// TIA Portal project "FactoryIO_Template_S7-1200_V15_V16" (V16)
// Vorlageprojekt für das Buch mit Zielsystem S7-1200

(* hardware
DEVICE "S7-1200-Station_1"  S7-1200 Station
   slot 0: "Baugruppenträger_0"  Rack  V1.0
   slot 1: "PLC_1"  CPU 1214C DC/DC/Rly  6ES7 214-1HG40-0XB0  V4.4
   slot 2: "DQ 16x24VDC_1"  SM 1222 DQ16 x 24VDC  6ES7 222-1BH32-0XB0  V2.0
   slot 3: "DQ 16x24VDC_2"  SM 1222 DQ16 x 24VDC  6ES7 222-1BH32-0XB0  V2.0
   slot 4: "DQ 16x24VDC_3"  SM 1222 DQ16 x 24VDC  6ES7 222-1BH32-0XB0  V2.0
   slot 5: "DQ 16x24VDC_4"  SM 1222 DQ16 x 24VDC  6ES7 222-1BH32-0XB0  V2.0
   slot 6: "DQ 16x24VDC_5"  SM 1222 DQ16 x 24VDC  6ES7 222-1BH32-0XB0  V2.0
   slot 7: "DQ 16x24VDC_6"  SM 1222 DQ16 x 24VDC  6ES7 222-1BH32-0XB0  V2.0
   slot 8: "DQ 16x24VDC_7"  SM 1222 DQ16 x 24VDC  6ES7 222-1BH32-0XB0  V2.0
   slot 9: "DQ 16x24VDC_8"  SM 1222 DQ16 x 24VDC  6ES7 222-1BH32-0XB0  V2.0
*)

// ===== PLC "PLC_1"  CPU 1214C DC/DC/Rly =====

VAR_GLOBAL   // PLC tag table "Standard-Variablentabelle"
   "System" AT %M0.0 : Bool;
   "Blue Lids at Place Memory" AT %M0.1 : Bool;
   "Blue Bases at Place Memory" AT %M0.2 : Bool;
   "Blue S1" AT %M0.3 : Bool;
   "Blue S2" AT %M0.4 : Bool;
   "Blue S3" AT %M0.5 : Bool;
   "Blue S4" AT %M0.6 : Bool;
   "Blue S5" AT %M0.7 : Bool;
   "Blue S6" AT %M1.0 : Bool;
   "Blue S7" AT %M1.1 : Bool;
   "Blue S8" AT %M1.2 : Bool;
   "Blue S9" AT %M1.3 : Bool;
   "Blue S10" AT %M1.4 : Bool;
   "Blue S11" AT %M1.5 : Bool;
   "Green Lid at place memory" AT %M2.0 : Bool;
   "Green bases at place memory" AT %M2.1 : Bool;
   "Green S1" AT %M2.2 : Bool;
   "Green S2" AT %M2.3 : Bool;
   "Green S3" AT %M2.4 : Bool;
   "Green S4" AT %M2.5 : Bool;
   "Green S5" AT %M2.6 : Bool;
   "Green S6" AT %M2.7 : Bool;
   "Green S7" AT %M3.0 : Bool;
   "Green S8" AT %M3.1 : Bool;
   "Green S9" AT %M3.2 : Bool;
   "Green S10" AT %M3.3 : Bool;
   "Green S11" AT %M3.4 : Bool;
   "Metal S1" AT %M3.5 : Bool;
   "Metal S2" AT %M3.6 : Bool;
   "Metal S3" AT %M3.7 : Bool;
   "Metal S4" AT %M4.0 : Bool;
   "Metal S5" AT %M4.1 : Bool;
   "Metal S6" AT %M4.2 : Bool;
   "Metal S7" AT %M4.3 : Bool;
   "Metal S8" AT %M4.4 : Bool;
   "Metal S9" AT %M4.5 : Bool;
   "Metal S10" AT %M4.6 : Bool;
   "Metal S11" AT %M4.7 : Bool;
   "Metal Lid at place memory" AT %M5.0 : Bool;
   "Metal bases at place memory" AT %M5.1 : Bool;
   "Blue Pallet lid at place memory" AT %M5.2 : Bool;
   "Blue Pallet bases at place memory" AT %M5.3 : Bool;
   "Blue Pallet S1" AT %M5.4 : Bool;
   "Blue Pallet S2" AT %M5.5 : Bool;
   "Blue Pallet S3" AT %M5.6 : Bool;
   "Blue Pallet S4" AT %M5.7 : Bool;
   "Blue Pallet S5" AT %M6.0 : Bool;
   "Blue Pallet S6" AT %M6.1 : Bool;
   "Blue Pallet S7" AT %M6.2 : Bool;
   "Blue Pallet S8" AT %M6.3 : Bool;
   "Blue Pallet S9" AT %M6.4 : Bool;
   "Blue Pallet S10" AT %M6.5 : Bool;
   "Blue Pallet S11" AT %M6.6 : Bool;
   "Green Pallet lid at place memory(1)" AT %M6.7 : Bool;
   "Green Pallet bases at place memory(1)" AT %M7.0 : Bool;
   "Green Pallet S1" AT %M7.1 : Bool;
   "Green Pallet S2" AT %M7.2 : Bool;
   "Green Pallet S3" AT %M7.3 : Bool;
   "Green Pallet S4" AT %M7.4 : Bool;
   "Green Pallet S5" AT %M7.5 : Bool;
   "Green  Pallet S6" AT %M7.6 : Bool;
   "Green  Pallet S7" AT %M7.7 : Bool;
   "Green Pallet S8" AT %M8.0 : Bool;
   "Green Pallet S9" AT %M8.1 : Bool;
   "Green Pallet S10" AT %M8.2 : Bool;
   "Green Pallet S11" AT %M8.3 : Bool;
   "Metal Pallet lid at place memory(2)" AT %M8.4 : Bool;
   "Metal Pallet bases at place memory(2)" AT %M8.5 : Bool;
   "Metal  Pallet S1" AT %M8.6 : Bool;
   "Metal Pallet S2" AT %M8.7 : Bool;
   "Metal Pallet S3" AT %M9.0 : Bool;
   "Metal Pallet S4" AT %M9.1 : Bool;
   "Metal Pallet S5" AT %M9.2 : Bool;
   "Metal Pallet S6" AT %M9.3 : Bool;
   "Metal Pallet S7" AT %M9.4 : Bool;
   "Metal Pallet S8" AT %M9.5 : Bool;
   "Metal Pallet S9" AT %M9.6 : Bool;
   "Metal Pallet S10" AT %M9.7 : Bool;
   "Metal Pallet S11" AT %M10.0 : Bool;
   "Blue Elevator S1" AT %M11.0 : Bool;
   "Blue Elevator Completed" AT %M11.2 : Bool;
   "Green Elevator S1" AT %M11.3 : Bool;
   "Green Elevator Completed" AT %M11.4 : Bool;
   "Metal Elevator S1" AT %M11.5 : Bool;
   "Metal Elevator Completed" AT %M11.6 : Bool;
   "Blue Elevator S2" AT %M11.7 : Bool;
   "Green Elevator S2" AT %M12.0 : Bool;
   "Metal Elevator S2" AT %M12.1 : Bool;
   "Blue Elevator S3" AT %M12.2 : Bool;
   "Green Elevator S3" AT %M12.3 : Bool;
   "Metal Elevator S3" AT %M12.4 : Bool;
   "Blue Turn Table Completed" AT %M13.5 : Bool;
   "Metal Turn Table Completed" AT %M13.4 : Bool;
   "Crane 1 S1" AT %M13.6 : Bool;
   "Crane 1 S2" AT %M13.7 : Bool;
   "Crane 1 S3" AT %M14.0 : Bool;
   "Crane 1 S4" AT %M14.1 : Bool;
   "Crane 1 S5" AT %M14.2 : Bool;
   "Crane 1 S6" AT %M14.3 : Bool;
   "Crane 1 S3 Positive Edge Mem" AT %M14.4 : Bool;
   "Turn Table Completed" AT %M14.5 : Bool;
   "Crane 2 Step 1" AT %M14.6 : Bool;
   "Crane 2 Step 2" AT %M14.7 : Bool;
   "Crane 2 Step 3" AT %M15.0 : Bool;
   "Crane 2 Step 4" AT %M15.1 : Bool;
   "Crane 2 Step 5" AT %M15.2 : Bool;
   "Crane 2 Step 6" AT %M15.3 : Bool;
   "Crane 2 P3 Pos Memory" AT %M15.4 : Bool;
   "Crane 3 Step 1" AT %M15.5 : Bool;
   "Crane 3 Step 2" AT %M15.6 : Bool;
   "Crane 3 Step 3" AT %M15.7 : Bool;
   "Crane 3 Step 4" AT %M16.0 : Bool;
   "Crane 3 Step 5" AT %M16.1 : Bool;
   "Crane 3 Step 6" AT %M16.2 : Bool;
   "Crane 3 P3 Pos Mem" AT %M16.3 : Bool;
   "Palletizer 1 Pallet Entry sensor" AT %I8.7 : Bool;
   "Palletizer 1 Move To Limit" AT %I12.7 : Bool;
   "Palletizer 1 S1" AT %M18.1 : Bool;
   "Box Entry Sensor Memory" AT %M18.2 : Bool;
   "Palletizer S2" AT %M18.3 : Bool;
   "Palletizer S3" AT %M18.4 : Bool;
   "Palletizer S4" AT %M18.5 : Bool;
   "Palletizer S5" AT %M18.6 : Bool;
END_VAR

VAR_GLOBAL   // PLC tag table "Tag table from XML_1"
   "Start All Factory" AT %I0.0 : Bool;
   "Stop All Factory" AT %I0.1 : Bool;
   "Emergency Factory" AT %I0.2 : Bool;
   "Blue Pusher Back Limit" AT %I0.3 : Bool;
   "Blue Pusher Front Limit" AT %I0.4 : Bool;
   "Green Pusher Front Limit" AT %I0.5 : Bool;
   "Green Pusher Back Limit" AT %I0.6 : Bool;
   "Metal Pusher Back Limit" AT %I0.7 : Bool;
   "Metal Pusher Front Limit" AT %I1.0 : Bool;
   "Blue Vision Sensor" AT %I1.1 : Bool;
   "Green Vision Sensor" AT %I1.2 : Bool;
   "Metal Vision Sensor" AT %I1.3 : Bool;
   "Blue Machine is Busy" AT %I1.4 : Bool;
   "Green Machine is Busy" AT %I1.5 : Bool;
   "Metal Machine is Busy" AT %I1.6 : Bool;
   "Blue Lid at Place" AT %I1.7 : Bool;
   "Blue base at place" AT %I2.0 : Bool;
   "Blue Bases Clamped" AT %I2.1 : Bool;
   "Blue Lid Clamped" AT %I2.2 : Bool;
   "Blue item detected" AT %I2.3 : Bool;
   "Green Lid at Place" AT %I2.4 : Bool;
   "Green Base at Place" AT %I2.5 : Bool;
   "Green Base Clamped" AT %I2.6 : Bool;
   "Green Item Detected" AT %I2.7 : Bool;
   "Green Lid Clamped" AT %I3.0 : Bool;
   "Metal Lid at Place" AT %I3.1 : Bool;
   "Metal Base at Place" AT %I3.2 : Bool;
   "Metal Base Clamped" AT %I3.3 : Bool;
   "Metal Lid Clamped" AT %I3.4 : Bool;
   "Metal Item Detected" AT %I3.5 : Bool;
   "Blue Pallet Base at Place" AT %I3.6 : Bool;
   "Blue Pallet Lid at Place" AT %I3.7 : Bool;
   "Blue Pallet Item Detected" AT %I4.0 : Bool;
   "Blue Pallet Lid Clamped" AT %I4.1 : Bool;
   "Green Pallet Base at Place" AT %I4.2 : Bool;
   "Green Pallet Item Detected" AT %I4.3 : Bool;
   "Green Pallet Lid at Place" AT %I4.4 : Bool;
   "Green Pallet Lid Clamped" AT %I4.5 : Bool;
   "Metal Pallet Base at Place" AT %I4.6 : Bool;
   "Metal Pallet Item Detected" AT %I4.7 : Bool;
   "Metal Pallet Lid at Place" AT %I5.0 : Bool;
   "Metal Pallet Lid Clamped" AT %I5.1 : Bool;
   "Call Blue Elevator" AT %I5.2 : Bool;
   "Call Green Elevator" AT %I5.3 : Bool;
   "Call Metal Elevator" AT %I5.4 : Bool;
   "Blue Turn Table Back Limit" AT %I5.5 : Bool;
   "Blue Turn Table Front Limit" AT %I5.6 : Bool;
   "Blue Turn Table Limit 0" AT %I5.7 : Bool;
   "Blue Turn Table Limit 90" AT %I6.0 : Bool;
   "Metal Turn Table Back  Limit" AT %I6.1 : Bool;
   "Metal Turn Table Front Limit" AT %I6.3 : Bool;
   "Metal Turn Table Limit 0" AT %I6.4 : Bool;
   "Metal Turn Table Limit 90" AT %I6.5 : Bool;
   "Crane 1 Moving X" AT %I6.6 : Bool;
   "Crane 1 Moving Z" AT %I6.7 : Bool;
   "Crane 1 At Load Sensor" AT %I7.0 : Bool;
   "Crane 1At Entry Sensor" AT %I7.1 : Bool;
   "Crane 2 Moving X" AT %I7.2 : Bool;
   "Crane 2 Moving Z" AT %I7.3 : Bool;
   "Crane 2 At Load Sensor" AT %I7.4 : Bool;
   "Crane 3 Moving X" AT %I7.6 : Bool;
   "Crane 3 Moving Z" AT %I7.7 : Bool;
   "Crane 3 At Load Sensor" AT %I8.0 : Bool;
   "Crane 3 At Entry Sensor" AT %I8.1 : Bool;
   "Palletizer 1 (Clamped)" AT %I8.2 : Bool;
   "Palletizer 1 Box Entry Sensor" AT %I8.3 : Bool;
   "Palletizer 1 (Pusher Limit)" AT %I8.4 : Bool;
   "Palletizer 1 (Elevator Moving)" AT %I8.5 : Bool;
   "Palletizer 1 Elevator (Front Limit)" AT %I8.6 : Bool;
   "Start Light Indicator" AT %Q0.0 : Bool;
   "Stop Light Indicator" AT %Q0.1 : Bool;
   "Starter Conveyor 1" AT %Q0.2 : Bool;
   "Starter Conveyor 2" AT %Q0.3 : Bool;
   "Starter Conveyor 3" AT %Q0.4 : Bool;
   "Starter Conveyor 4" AT %Q0.5 : Bool;
   "Starter Conveyor 5" AT %Q0.6 : Bool;
   "Blue Entry Conveyor" AT %Q0.7 : Bool;
   "Green Entry Conveyor" AT %Q1.0 : Bool;
   "Metal Entry Conveyor" AT %Q1.1 : Bool;
   "Blue Pusher" AT %Q1.2 : Bool;
   "Green Pusher" AT %Q1.3 : Bool;
   "Metal Pusher" AT %Q1.4 : Bool;
   "Blue Machine Start" AT %Q1.5 : Bool;
   "Green Machine Start" AT %Q1.6 : Bool;
   "Metal Machine Start" AT %Q1.7 : Bool;
   "Blue Product Emitter" AT %Q2.0 : Bool;
   "Green Product Emitter" AT %Q2.1 : Bool;
   "Metal Product Emitter" AT %Q2.2 : Bool;
   "Blue Lids Conveyor" AT %Q2.3 : Bool;
   "Blue Bases Conveyor" AT %Q2.4 : Bool;
   "Blue Clamp Lid" AT %Q2.5 : Bool;
   "Blue Clamp Bases" AT %Q2.6 : Bool;
   "Blue Move Z" AT %Q2.7 : Bool;
   "Blue Move X" AT %Q3.0 : Bool;
   "Blue Grab" AT %Q3.1 : Bool;
   "Blue pos raise bases" AT %Q3.2 : Bool;
   "Blue pos raise lids" AT %Q3.3 : Bool;
   "Green Lid Conveyor" AT %Q3.4 : Bool;
   "Green Base Conveyor" AT %Q3.5 : Bool;
   "Green Clamp Lid" AT %Q3.6 : Bool;
   "Green Clamp Base" AT %Q3.7 : Bool;
   "Green Move Z" AT %Q4.0 : Bool;
   "Green Move X" AT %Q4.1 : Bool;
   "Green Grab" AT %Q4.2 : Bool;
   "Green pos raise lids" AT %Q4.3 : Bool;
   "Green pos raise bases" AT %Q4.4 : Bool;
   "Metal Lids Conveyor" AT %Q4.5 : Bool;
   "Metal Bases Conveyor" AT %Q4.6 : Bool;
   "Metal Clamp Lid" AT %Q4.7 : Bool;
   "Metal Clamp Base" AT %Q5.0 : Bool;
   "Metal Move Z" AT %Q5.1 : Bool;
   "Metal Move X" AT %Q5.2 : Bool;
   "Metal Grab" AT %Q5.3 : Bool;
   "Metal pos raise base" AT %Q5.4 : Bool;
   "Metal pos raise lids" AT %Q5.5 : Bool;
   "Blue Pallet Base Conveyor" AT %Q5.6 : Bool;
   "Blue Pallet Grab" AT %Q5.7 : Bool;
   "Blue Pallet Lid Clamp" AT %Q6.0 : Bool;
   "Blue Pallet Lid Conveyor" AT %Q6.1 : Bool;
   "Blue Pallet pos raise lid" AT %Q6.2 : Bool;
   "Blue Pallet Move X" AT %Q6.3 : Bool;
   "Blue Pallet Move Z" AT %Q6.4 : Bool;
   "Green Pallet Base Conveyor" AT %Q6.5 : Bool;
   "Green Pallet Grab" AT %Q6.6 : Bool;
   "Green Pallet Lid Clamp" AT %Q6.7 : Bool;
   "Green Pallet Lid Conveyor" AT %Q7.0 : Bool;
   "Green Pallet Move X" AT %Q7.1 : Bool;
   "Green Pallet Move Z" AT %Q7.2 : Bool;
   "Green Pallet pos raise lid" AT %Q7.3 : Bool;
   "Metal Pallet Base Conveyor" AT %Q7.4 : Bool;
   "Metal Pallet Grab" AT %Q7.5 : Bool;
   "Metal Pallet Lid Clamp" AT %Q7.6 : Bool;
   "Metal Pallet Lid Conveyor" AT %Q7.7 : Bool;
   "Metal Pallet Move X" AT %Q8.0 : Bool;
   "Metal Pallet Move Z" AT %Q8.1 : Bool;
   "Metal Pallet pos raise lid" AT %Q8.2 : Bool;
   "Blue Elevator Roller" AT %Q8.3 : Bool;
   "Green Elevator Roller" AT %Q8.4 : Bool;
   "Metal Elevator Roller" AT %Q8.5 : Bool;
   "Blue Turn Table Roll +" AT %Q8.6 : Bool;
   "Blue Turn Table Roll -" AT %Q8.7 : Bool;
   "Blue Turn Table Turn" AT %Q9.0 : Bool;
   "Metal Turn Table Roll +" AT %Q9.1 : Bool;
   "Metal Turn Table Roll -" AT %Q9.2 : Bool;
   "Metal Turn Table Turn" AT %Q9.3 : Bool;
   "Crane 1 Left" AT %Q9.4 : Bool;
   "Crane 1 Lift" AT %Q9.5 : Bool;
   "Crane 1 Right" AT %Q9.6 : Bool;
   "Crane 1 Entry Conveyor" AT %Q9.7 : Bool;
   "Crane 1 Loading Conveyor" AT %Q10.0 : Bool;
   "Crane 2 Lift" AT %Q10.1 : Bool;
   "Crane 2 Left" AT %Q10.2 : Bool;
   "Crane 2 Right" AT %Q10.3 : Bool;
   "Crane 2 Loading Conveyor" AT %Q10.5 : Bool;
   "Crane 3 Left" AT %Q10.6 : Bool;
   "Crane 3 Lift" AT %Q10.7 : Bool;
   "Crane 3 Right" AT %Q11.0 : Bool;
   "Crane 3 Entry Conveyor" AT %Q11.1 : Bool;
   "Crane 3 Loading Conveyor" AT %Q11.2 : Bool;
   "Green Conveyor 1" AT %Q11.3 : Bool;
   "Green Conveyor 2" AT %Q11.4 : Bool;
   "Palletizer 1 (Push)" AT %Q11.5 : Bool;
   "Palletizer 1 (Turn)" AT %Q11.6 : Bool;
   "Palletizer 1 (Clamp)" AT %Q11.7 : Bool;
   "Palletizer 1 Chain (+)" AT %Q12.0 : Bool;
   "Palletizer 1 Elevator (+)" AT %Q12.1 : Bool;
   "Palletizer 1 Elevator (-)" AT %Q12.2 : Bool;
   "Palletizer 3 (Open Plate)" AT %Q12.3 : Bool;
   "Palletizer 1 Box Entry Conveyor" AT %Q12.4 : Bool;
   "Palletizer 1 Pallet Entry Conveyor" AT %Q12.5 : Bool;
   "Palletizer 1 Belt (+)" AT %Q12.6 : Bool;
   "Blue Elevator Set Point" AT %QD16 : Real;
   "Green Elevator Set Point" AT %QD20 : Real;
   "Metal Elevator Set Point" AT %QD24 : Real;
   "Crane 1 Target Position" AT %QD28 : DInt;
   "Crane 2 Target Position" AT %QD32 : DInt;
   "Crane 3 Target Position" AT %QD36 : DInt;
END_VAR

DATA_BLOCK "Blue Pallet PP"   // DB1
{ S7_Optimized_Access := 'TRUE' }
VERSION : 0.1
// stored: InstanceOfName Pick and Place
"Pick and Place"
BEGIN
END_DATA_BLOCK

DATA_BLOCK "Green Pallet PP"   // DB2
{ S7_Optimized_Access := 'TRUE' }
VERSION : 0.1
// stored: InstanceOfName Pick and Place
"Pick and Place"
BEGIN
END_DATA_BLOCK

DATA_BLOCK "Metal Pallet PP"   // DB3
{ S7_Optimized_Access := 'TRUE' }
VERSION : 0.1
// stored: InstanceOfName Pick and Place
"Pick and Place"
BEGIN
END_DATA_BLOCK

DATA_BLOCK "Blue Turn Table Right"   // DB4
{ S7_Optimized_Access := 'TRUE' }
VERSION : 0.1
// stored: InstanceOfName Turn Table Left
"Turn Table Left"
BEGIN
END_DATA_BLOCK

DATA_BLOCK "Blue Elevator"   // DB5
{ S7_Optimized_Access := 'TRUE' }
VERSION : 0.1
// stored: InstanceOfName Elevator
"Elevator"
BEGIN
END_DATA_BLOCK

DATA_BLOCK "Green Elevator"   // DB6
{ S7_Optimized_Access := 'TRUE' }
VERSION : 0.1
// stored: InstanceOfName Elevator
"Elevator"
BEGIN
END_DATA_BLOCK

DATA_BLOCK "Metal Elevator"   // DB7
{ S7_Optimized_Access := 'TRUE' }
VERSION : 0.1
// stored: InstanceOfName Elevator
"Elevator"
BEGIN
END_DATA_BLOCK

DATA_BLOCK "Crane 1"   // DB8
{ S7_Optimized_Access := 'TRUE' }
VERSION : 0.1
// stored: InstanceOfName Stacker_Crane
"Stacker_Crane"
BEGIN
END_DATA_BLOCK

DATA_BLOCK "Pick and Place_DB"   // DB9
{ S7_Optimized_Access := 'TRUE' }
VERSION : 0.1
// stored: InstanceOfName Pick and Place
"Pick and Place"
BEGIN
END_DATA_BLOCK

DATA_BLOCK "Blue Lid and Bases PAP"   // DB10
{ S7_Optimized_Access := 'TRUE' }
VERSION : 0.1
// stored: InstanceOfName Pick and Place
"Pick and Place"
BEGIN
END_DATA_BLOCK

DATA_BLOCK "Green Lid and Base PAP"   // DB11
{ S7_Optimized_Access := 'TRUE' }
VERSION : 0.1
// stored: InstanceOfName Pick and Place
"Pick and Place"
BEGIN
END_DATA_BLOCK

DATA_BLOCK "Pick and Place_DB_1"   // DB12
{ S7_Optimized_Access := 'TRUE' }
VERSION : 0.1
// stored: InstanceOfName Pick and Place
"Pick and Place"
BEGIN
END_DATA_BLOCK

DATA_BLOCK "Metal Turn Table"   // DB13
{ S7_Optimized_Access := 'TRUE' }
VERSION : 0.1
// stored: InstanceOfName Turn Table Left
"Turn Table Left"
BEGIN
END_DATA_BLOCK

DATA_BLOCK "Blue Pallet Transfer Turn Table"   // DB14
{ S7_Optimized_Access := 'TRUE' }
VERSION : 0.1
// stored: InstanceOfName Turn Table Left
"Turn Table Left"
BEGIN
END_DATA_BLOCK

DATA_BLOCK "Turn Table Right_DB"   // DB15
{ S7_Optimized_Access := 'TRUE' }
VERSION : 0.1
// stored: InstanceOfName Turn Table Right
"Turn Table Right"
BEGIN
END_DATA_BLOCK

DATA_BLOCK "Metal Turn Table Right"   // DB17
{ S7_Optimized_Access := 'TRUE' }
VERSION : 0.1
// stored: InstanceOfName Turn Table Right
"Turn Table Right"
BEGIN
END_DATA_BLOCK

DATA_BLOCK "Blue Turn Table Left"   // DB18
{ S7_Optimized_Access := 'TRUE' }
VERSION : 0.1
// stored: InstanceOfName Turn Table Left
"Turn Table Left"
BEGIN
END_DATA_BLOCK

DATA_BLOCK "Crane 2"   // DB19
{ S7_Optimized_Access := 'TRUE' }
VERSION : 0.1
// stored: InstanceOfName Stacker_Crane
"Stacker_Crane"
BEGIN
END_DATA_BLOCK

DATA_BLOCK "Crane 3"   // DB20
{ S7_Optimized_Access := 'TRUE' }
VERSION : 0.1
// stored: InstanceOfName Stacker_Crane
"Stacker_Crane"
BEGIN
END_DATA_BLOCK

DATA_BLOCK "Palletizer_DB"   // DB24
{ S7_Optimized_Access := 'TRUE' }
VERSION : 0.1
// stored: InstanceOfName Palletizer
"Palletizer"
BEGIN
END_DATA_BLOCK

// folder: System blocks/Program resources

DATA_BLOCK "IEC_Timer_0_DB"   // DB16
{ S7_Optimized_Access := 'TRUE' }
AUTHOR : Simatic
FAMILY : IEC
NAME : IEC_TMR
VERSION : 1.0
// stored: InstanceOfName IEC_TIMER
"IEC_TIMER"
BEGIN
END_DATA_BLOCK

DATA_BLOCK "IEC_Counter_0_DB_1"   // DB23
{ S7_Optimized_Access := 'TRUE' }
AUTHOR : Simatic
FAMILY : IEC
NAME : CNTR
VERSION : 1.0
// stored: InstanceOfName IEC_COUNTER
"IEC_COUNTER"
BEGIN
END_DATA_BLOCK

// folder: (top level)

FUNCTION_BLOCK "Pick and Place"   // FB1, LAD
{ S7_Optimized_Access := 'TRUE' }
VERSION : 0.1
   VAR_INPUT
      System : Bool;
      Start : Bool;
      "Lid at place" : Bool;
      "Base at place" : Bool;
      "Lid Clamped" : Bool;
      "Base Clamped" : Bool;
      "Item Detected" : Bool;
   END_VAR
   VAR_OUTPUT
      "Lids Conveyor" : Bool;
      "Bases Conveyor" : Bool;
      "Lids at Place Memory" : Bool;
      "Bases at Place Memory" : Bool;
      "Clamp Lid" : Bool;
      "Clamp base" : Bool;
      "Move Z" : Bool;
      "Move X" : Bool;
      Grab : Bool;
      "Pos. raise bases" : Bool;
      "Pos. raise lids" : Bool;
      s1 : Bool;
      s2 : Bool;
      s3 : Bool;
      s4 : Bool;
      s5 : Bool;
      s6 : Bool;
      s7 : Bool;
      s8 : Bool;
      s9 : Bool;
      s10 : Bool;
      s11 : Bool;
   END_VAR
   VAR
      IEC_Timer_0_Instance : TON_TIME;
      IEC_Timer_0_Instance_1 : TON_TIME;
      IEC_Timer_0_Instance_2 : TON_TIME;
      IEC_Timer_0_Instance_3 : TON_TIME;
      IEC_Timer_0_Instance_4 : TON_TIME;
      IEC_Timer_0_Instance_5 : TON_TIME;
      IEC_Timer_0_Instance_6 : TON_TIME;
      IEC_Timer_0_Instance_7 : TON_TIME;
   END_VAR
   VAR_TEMP   // added for the SCL form of the ladder/FBD networks
      _w1 : Bool;
   END_VAR
BEGIN

REGION Network 1: Opening Conveyors
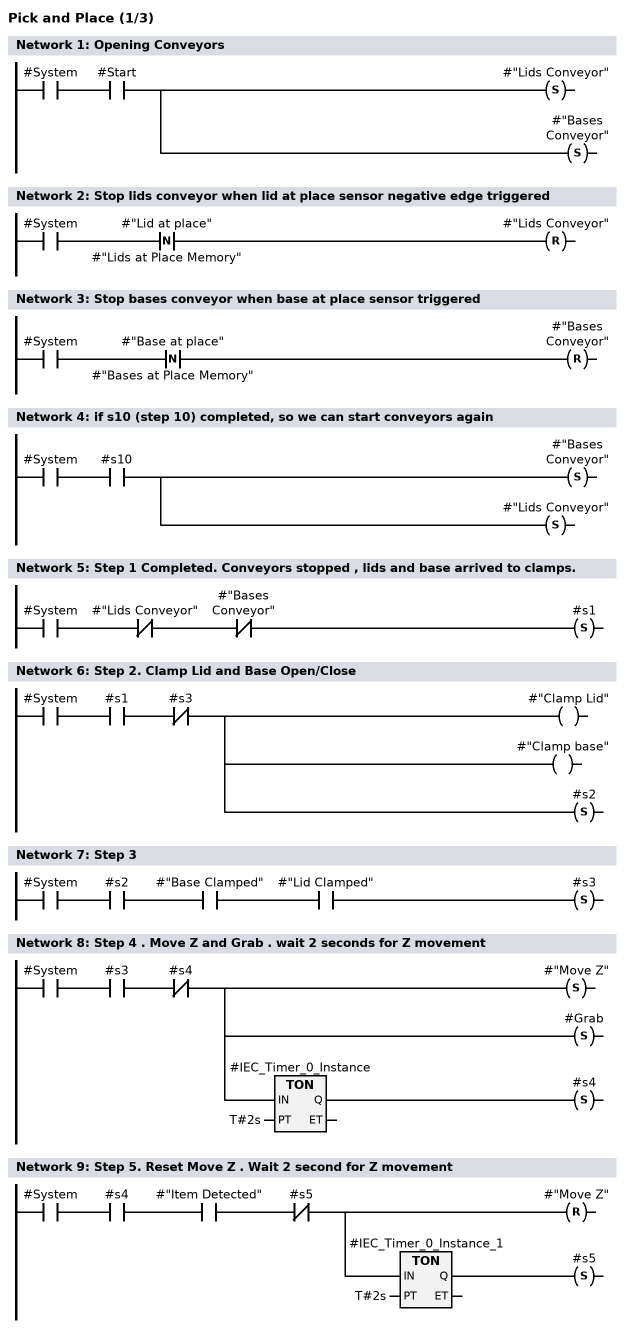
   RUNG wire#powerrail
      Contact( #System )
      Contact( #Start )
      wire#w1
      S_Coil( #"Lids Conveyor" )
   END_RUNG
   RUNG wire#w1
      S_Coil( #"Bases Conveyor" )
   END_RUNG
   // the same network as SCL:
   IF #System AND #Start THEN
       #"Lids Conveyor" := TRUE;
       #"Bases Conveyor" := TRUE;
   END_IF;
END_REGION

REGION Network 2: Stop lids conveyor when lid at place sensor negative edge triggered
   RUNG wire#powerrail
      Contact( #System )
      N_Contact(operand := #"Lid at place", bit := #"Lids at Place Memory")
      R_Coil( #"Lids Conveyor" )
   END_RUNG
   // the same network as SCL:
   #_w1 := #System AND NOT #"Lid at place" AND #"Lids at Place Memory";   // falling edge of #"Lid at place"
   #"Lids at Place Memory" := #"Lid at place";
   IF #_w1 THEN #"Lids Conveyor" := FALSE; END_IF;
END_REGION

REGION Network 3: Stop bases conveyor when base at place sensor triggered
   RUNG wire#powerrail
      Contact( #System )
      N_Contact(operand := #"Base at place", bit := #"Bases at Place Memory")
      R_Coil( #"Bases Conveyor" )
   END_RUNG
   // the same network as SCL:
   #_w1 := #System AND NOT #"Base at place" AND #"Bases at Place Memory";   // falling edge of #"Base at place"
   #"Bases at Place Memory" := #"Base at place";
   IF #_w1 THEN #"Bases Conveyor" := FALSE; END_IF;
END_REGION

REGION Network 4: if s10 (step 10) completed, so we can start conveyors again
   RUNG wire#powerrail
      Contact( #System )
      Contact( #s10 )
      wire#w1
      S_Coil( #"Bases Conveyor" )
   END_RUNG
   RUNG wire#w1
      S_Coil( #"Lids Conveyor" )
   END_RUNG
   // the same network as SCL:
   IF #System AND #s10 THEN
       #"Bases Conveyor" := TRUE;
       #"Lids Conveyor" := TRUE;
   END_IF;
END_REGION

REGION Network 5: Step 1 Completed. Conveyors stopped , lids and base arrived to clamps.
   RUNG wire#powerrail
      Contact( #System )
      I_Contact( #"Lids Conveyor" )
      I_Contact( #"Bases Conveyor" )
      S_Coil( #s1 )
   END_RUNG
   // the same network as SCL:
   IF #System AND NOT #"Lids Conveyor" AND NOT #"Bases Conveyor" THEN #s1 := TRUE; END_IF;
END_REGION

REGION Network 6: Step 2. Clamp Lid and Base Open/Close
   RUNG wire#powerrail
      Contact( #System )
      Contact( #s1 )
      I_Contact( #s3 )
      wire#w1
      Coil( #"Clamp Lid" )
   END_RUNG
   RUNG wire#w1
      Coil( #"Clamp base" )
   END_RUNG
   RUNG wire#w1
      S_Coil( #s2 )
   END_RUNG
   // the same network as SCL:
   #"Clamp Lid" := #System AND #s1 AND NOT #s3;
   #"Clamp base" := #"Clamp Lid";
   IF #"Clamp Lid" THEN #s2 := TRUE; END_IF;
END_REGION

REGION Network 7: Step 3
   RUNG wire#powerrail
      Contact( #System )
      Contact( #s2 )
      Contact( #"Base Clamped" )
      Contact( #"Lid Clamped" )
      S_Coil( #s3 )
   END_RUNG
   // the same network as SCL:
   IF #System AND #s2 AND #"Base Clamped" AND #"Lid Clamped" THEN #s3 := TRUE; END_IF;
END_REGION

REGION Network 8: Step 4 . Move Z and Grab . wait 2 seconds for Z movement
   #_w1 := #System AND #s3 AND NOT #s4;
   IF #_w1 THEN
       #"Move Z" := TRUE;
       #Grab := TRUE;
   END_IF;
   #IEC_Timer_0_Instance(IN := #_w1, PT := T#2s);   // TON
   IF #IEC_Timer_0_Instance.Q THEN #s4 := TRUE; END_IF;
END_REGION

REGION Network 9: Step 5. Reset Move Z . Wait 2 second for Z movement
   #_w1 := #System AND #s4 AND #"Item Detected" AND NOT #s5;
   IF #_w1 THEN #"Move Z" := FALSE; END_IF;
   #IEC_Timer_0_Instance_1(IN := #_w1, PT := T#2s);   // TON
   IF #IEC_Timer_0_Instance_1.Q THEN #s5 := TRUE; END_IF;
END_REGION

REGION Network 10: Step 6 Move X. Wait 2 seconds for X movement
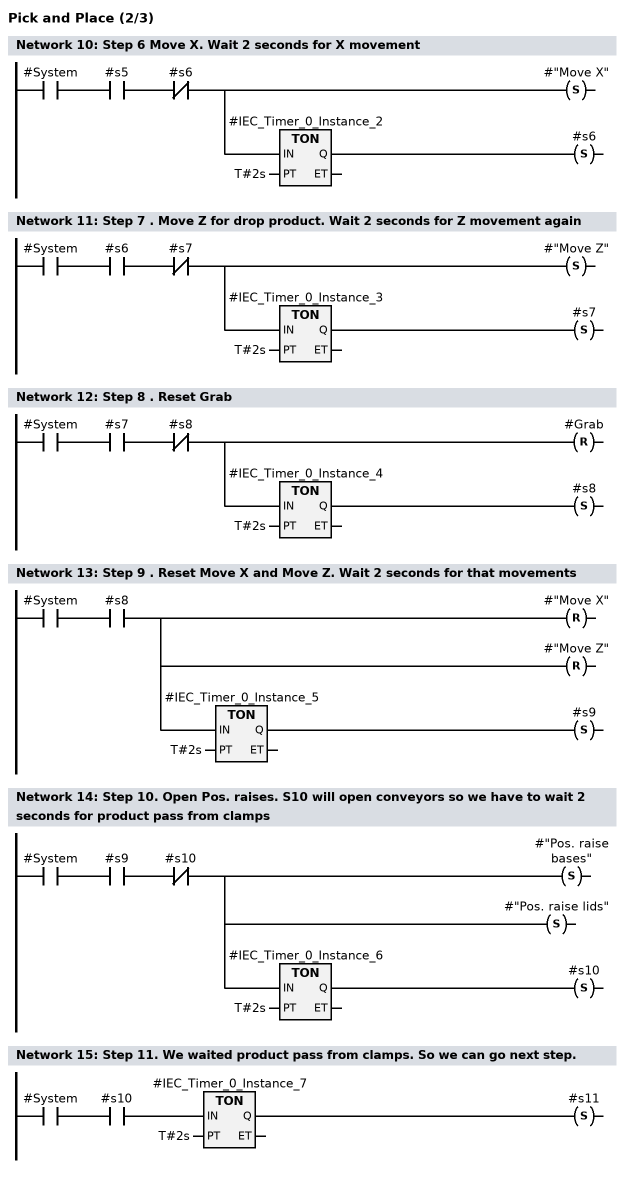
   #_w1 := #System AND #s5 AND NOT #s6;
   IF #_w1 THEN #"Move X" := TRUE; END_IF;
   #IEC_Timer_0_Instance_2(IN := #_w1, PT := T#2s);   // TON
   IF #IEC_Timer_0_Instance_2.Q THEN #s6 := TRUE; END_IF;
END_REGION

REGION Network 11: Step 7 . Move Z for drop product. Wait 2 seconds for Z movement again
   #_w1 := #System AND #s6 AND NOT #s7;
   IF #_w1 THEN #"Move Z" := TRUE; END_IF;
   #IEC_Timer_0_Instance_3(IN := #_w1, PT := T#2s);   // TON
   IF #IEC_Timer_0_Instance_3.Q THEN #s7 := TRUE; END_IF;
END_REGION

REGION Network 12: Step 8 . Reset Grab
   #_w1 := #System AND #s7 AND NOT #s8;
   IF #_w1 THEN #Grab := FALSE; END_IF;
   #IEC_Timer_0_Instance_4(IN := #_w1, PT := T#2s);   // TON
   IF #IEC_Timer_0_Instance_4.Q THEN #s8 := TRUE; END_IF;
END_REGION

REGION Network 13: Step 9 . Reset Move X and Move Z. Wait 2 seconds for that movements
   #_w1 := #System AND #s8;
   IF #_w1 THEN
       #"Move X" := FALSE;
       #"Move Z" := FALSE;
   END_IF;
   #IEC_Timer_0_Instance_5(IN := #_w1, PT := T#2s);   // TON
   IF #IEC_Timer_0_Instance_5.Q THEN #s9 := TRUE; END_IF;
END_REGION

REGION Network 14: Step 10. Open Pos. raises. S10 will open conveyors so we have to wait 2 seconds for product pass from clamps
   #_w1 := #System AND #s9 AND NOT #s10;
   IF #_w1 THEN
       #"Pos. raise bases" := TRUE;
       #"Pos. raise lids" := TRUE;
   END_IF;
   #IEC_Timer_0_Instance_6(IN := #_w1, PT := T#2s);   // TON
   IF #IEC_Timer_0_Instance_6.Q THEN #s10 := TRUE; END_IF;
END_REGION

REGION Network 15: Step 11. We waited product pass from clamps. So we can go next step.
   #IEC_Timer_0_Instance_7(IN := #System AND #s10, PT := T#2s);   // TON
   IF #IEC_Timer_0_Instance_7.Q THEN #s11 := TRUE; END_IF;
END_REGION

REGION Network 16: Pick and Place all movements completed. So we can reset all memories for loop.
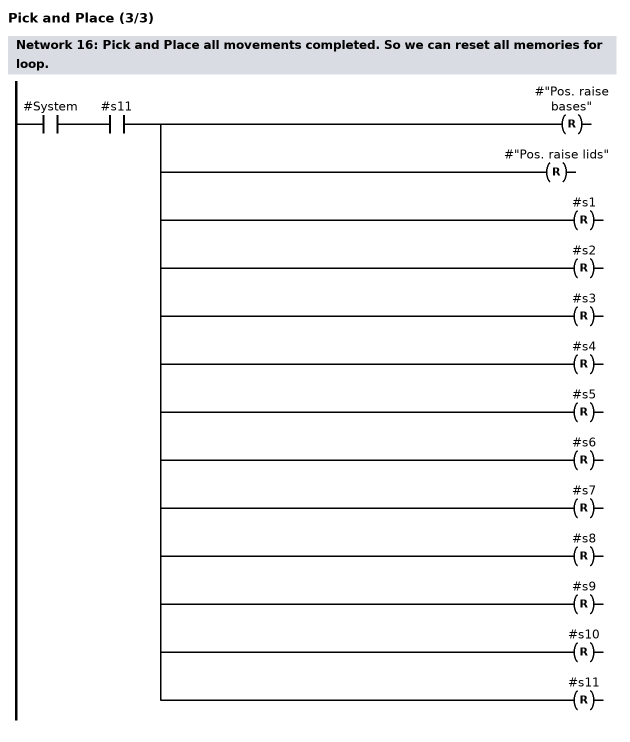
   RUNG wire#powerrail
      Contact( #System )
      Contact( #s11 )
      wire#w1
      R_Coil( #"Pos. raise bases" )
   END_RUNG
   RUNG wire#w1
      R_Coil( #"Pos. raise lids" )
   END_RUNG
   RUNG wire#w1
      R_Coil( #s1 )
   END_RUNG
   RUNG wire#w1
      R_Coil( #s2 )
   END_RUNG
   RUNG wire#w1
      R_Coil( #s3 )
   END_RUNG
   RUNG wire#w1
      R_Coil( #s4 )
   END_RUNG
   RUNG wire#w1
      R_Coil( #s5 )
   END_RUNG
   RUNG wire#w1
      R_Coil( #s6 )
   END_RUNG
   RUNG wire#w1
      R_Coil( #s7 )
   END_RUNG
   RUNG wire#w1
      R_Coil( #s8 )
   END_RUNG
   RUNG wire#w1
      R_Coil( #s9 )
   END_RUNG
   RUNG wire#w1
      R_Coil( #s10 )
   END_RUNG
   RUNG wire#w1
      R_Coil( #s11 )
   END_RUNG
   // the same network as SCL:
   IF #System AND #s11 THEN
       #"Pos. raise bases" := FALSE;
       #"Pos. raise lids" := FALSE;
       #s1 := FALSE;
       #s2 := FALSE;
       #s3 := FALSE;
       #s4 := FALSE;
       #s5 := FALSE;
       #s6 := FALSE;
       #s7 := FALSE;
       #s8 := FALSE;
       #s9 := FALSE;
       #s10 := FALSE;
       #s11 := FALSE;
   END_IF;
END_REGION
END_FUNCTION_BLOCK

FUNCTION_BLOCK "Elevator"   // FB2, LAD
{ S7_Optimized_Access := 'TRUE' }
VERSION : 0.1
   VAR_INPUT
      "Call Elevator" : Bool;
      System : Bool;
   END_VAR
   VAR_OUTPUT
      "Elevator Set Point" : Real;
      "Elevator Roller" : Bool;
      "Elevator Completed" : Bool;
      "Elevator S1" : Bool;
      "Elevator S2" : Bool;
      "Elevator S3" : Bool;
   END_VAR
   VAR
      IEC_Timer_0_Instance : TON_TIME;
      IEC_Timer_0_Instance_1 : TON_TIME;
      IEC_Timer_0_Instance_2 : TON_TIME;
   END_VAR
   VAR_TEMP   // added for the SCL form of the ladder/FBD networks
      _w1 : Bool;
   END_VAR
BEGIN

REGION Network 1: Pallet is coming. Elevator will go 2.1 position and roller will open
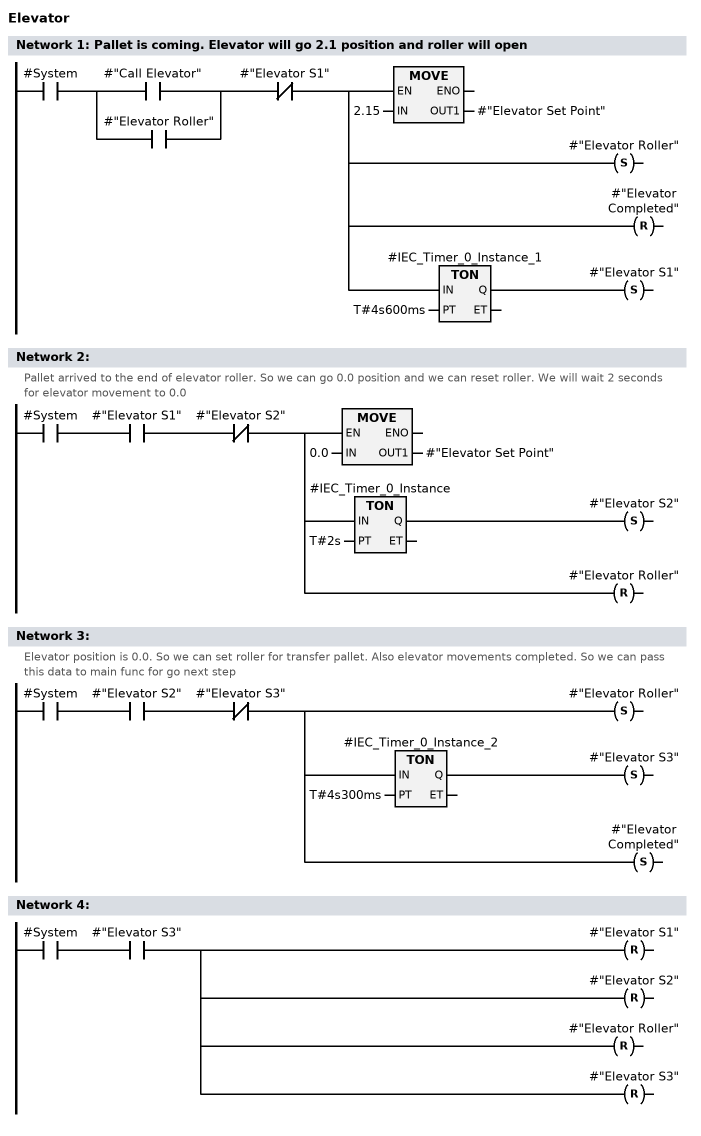
   #_w1 := #System AND (#"Call Elevator" OR #"Elevator Roller") AND NOT #"Elevator S1";
   IF #_w1 THEN
       #"Elevator Set Point" := 2.15;
       #"Elevator Roller" := TRUE;
       #"Elevator Completed" := FALSE;
   END_IF;
   #IEC_Timer_0_Instance_1(IN := #_w1, PT := T#4s600ms);   // TON
   IF #IEC_Timer_0_Instance_1.Q THEN #"Elevator S1" := TRUE; END_IF;
END_REGION

REGION Network 2
   // Pallet arrived to the end of elevator roller. So we can go 0.0 position and we can reset roller. We will wait 2 seconds for elevator movement to 0.0
   #_w1 := #System AND #"Elevator S1" AND NOT #"Elevator S2";
   IF #_w1 THEN #"Elevator Set Point" := 0.0; END_IF;
   #IEC_Timer_0_Instance(IN := #_w1, PT := T#2s);   // TON
   IF #IEC_Timer_0_Instance.Q THEN #"Elevator S2" := TRUE; END_IF;
   IF #_w1 THEN #"Elevator Roller" := FALSE; END_IF;
END_REGION

REGION Network 3
   // Elevator position is 0.0. So we can set roller for transfer pallet. Also elevator movements completed. So we can pass this data to main func for go next step
   #_w1 := #System AND #"Elevator S2" AND NOT #"Elevator S3";
   IF #_w1 THEN #"Elevator Roller" := TRUE; END_IF;
   #IEC_Timer_0_Instance_2(IN := #_w1, PT := T#4s300ms);   // TON
   IF #IEC_Timer_0_Instance_2.Q THEN #"Elevator S3" := TRUE; END_IF;
   IF #_w1 THEN #"Elevator Completed" := TRUE; END_IF;
END_REGION

REGION Network 4
   RUNG wire#powerrail
      Contact( #System )
      Contact( #"Elevator S3" )
      wire#w1
      R_Coil( #"Elevator S1" )
   END_RUNG
   RUNG wire#w1
      R_Coil( #"Elevator S2" )
   END_RUNG
   RUNG wire#w1
      R_Coil( #"Elevator Roller" )
   END_RUNG
   RUNG wire#w1
      R_Coil( #"Elevator S3" )
   END_RUNG
   // the same network as SCL:
   IF #System AND #"Elevator S3" THEN
       #"Elevator S1" := FALSE;
       #"Elevator S2" := FALSE;
       #"Elevator Roller" := FALSE;
       #"Elevator S3" := FALSE;
   END_IF;
END_REGION
END_FUNCTION_BLOCK

FUNCTION_BLOCK "Turn Table Left"   // FB3, LAD
{ S7_Optimized_Access := 'TRUE' }
VERSION : 0.1
   VAR_INPUT
      system : Bool;
      "Elevator Completed" : Bool;
      "Turn Table Front Limit" : Bool;
      "Turn Table Limit 0" : Bool;
      "Turn Table Limit 90" : Bool;
   END_VAR
   VAR_OUTPUT
      "Turn Table Input Roll" : Bool;
      "Turn Table Exit Roll" : Bool;
      "Turn Table Turn" : Bool;
      "Turn Table Completed" : Bool;
      "Turn Table is Busy" : Bool;
   END_VAR
   VAR
      IEC_Timer_0_Instance : TON_TIME;
   END_VAR
   VAR_TEMP   // added for the SCL form of the ladder/FBD networks
      _w1 : Bool;
   END_VAR
BEGIN

REGION Network 1: start turn table roll when elevator movements completed. and stop it when front limit sensor triggered
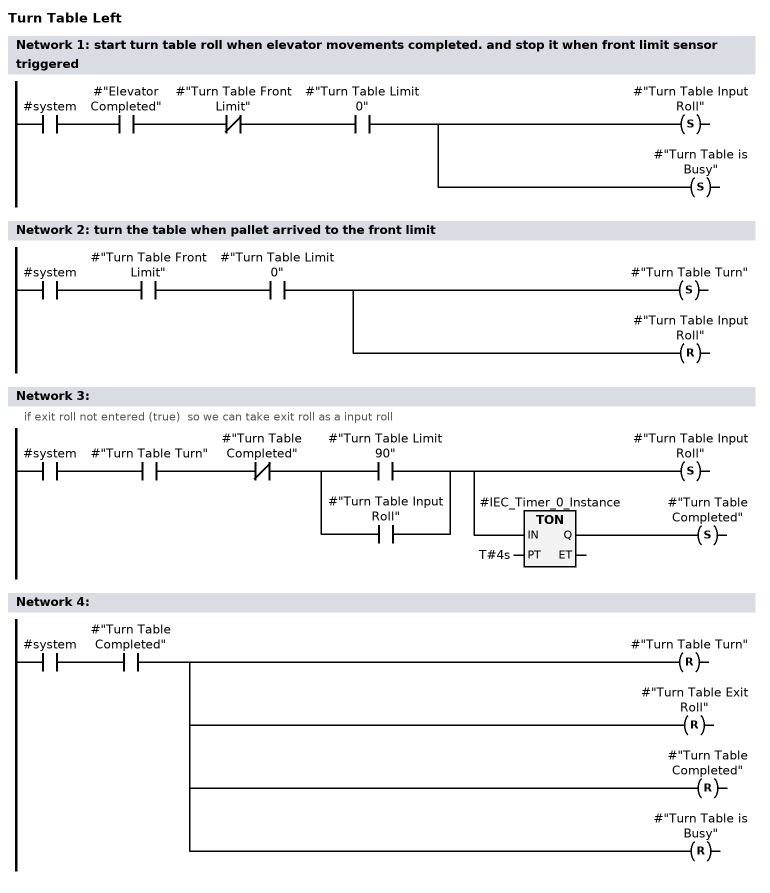
   RUNG wire#powerrail
      Contact( #system )
      Contact( #"Elevator Completed" )
      I_Contact( #"Turn Table Front Limit" )
      Contact( #"Turn Table Limit 0" )
      wire#w1
      S_Coil( #"Turn Table Input Roll" )
   END_RUNG
   RUNG wire#w1
      S_Coil( #"Turn Table is Busy" )
   END_RUNG
   // the same network as SCL:
   IF #system AND #"Elevator Completed" AND NOT #"Turn Table Front Limit" AND #"Turn Table Limit 0" THEN
       #"Turn Table Input Roll" := TRUE;
       #"Turn Table is Busy" := TRUE;
   END_IF;
END_REGION

REGION Network 2: turn the table when pallet arrived to the front limit
   RUNG wire#powerrail
      Contact( #system )
      Contact( #"Turn Table Front Limit" )
      Contact( #"Turn Table Limit 0" )
      wire#w1
      S_Coil( #"Turn Table Turn" )
   END_RUNG
   RUNG wire#w1
      R_Coil( #"Turn Table Input Roll" )
   END_RUNG
   // the same network as SCL:
   IF #system AND #"Turn Table Front Limit" AND #"Turn Table Limit 0" THEN
       #"Turn Table Turn" := TRUE;
       #"Turn Table Input Roll" := FALSE;
   END_IF;
END_REGION

REGION Network 3
   // if exit roll not entered (true)  so we can take exit roll as a input roll
   #_w1 := #system AND #"Turn Table Turn" AND NOT #"Turn Table Completed" AND (#"Turn Table Limit 90" OR #"Turn Table Input Roll");
   IF #_w1 THEN #"Turn Table Input Roll" := TRUE; END_IF;
   #IEC_Timer_0_Instance(IN := #_w1, PT := T#4s);   // TON
   IF #IEC_Timer_0_Instance.Q THEN #"Turn Table Completed" := TRUE; END_IF;
END_REGION

REGION Network 4
   RUNG wire#powerrail
      Contact( #system )
      Contact( #"Turn Table Completed" )
      wire#w1
      R_Coil( #"Turn Table Turn" )
   END_RUNG
   RUNG wire#w1
      R_Coil( #"Turn Table Exit Roll" )
   END_RUNG
   RUNG wire#w1
      R_Coil( #"Turn Table Completed" )
   END_RUNG
   RUNG wire#w1
      R_Coil( #"Turn Table is Busy" )
   END_RUNG
   // the same network as SCL:
   IF #system AND #"Turn Table Completed" THEN
       #"Turn Table Turn" := FALSE;
       #"Turn Table Exit Roll" := FALSE;
   END_IF;
   #_w1 := #system AND #"Turn Table Completed";
   IF #_w1 THEN
       #"Turn Table Completed" := FALSE;
       #"Turn Table is Busy" := FALSE;
   END_IF;
END_REGION
END_FUNCTION_BLOCK

FUNCTION_BLOCK "Stacker_Crane"   // FB4, LAD
{ S7_Optimized_Access := 'TRUE' }
VERSION : 0.1
   VAR_INPUT
      "At Entry" : Bool;
      "At Load" : Bool;
      "Moving Z" : Bool;
      "Moving X" : Bool;
      System : Bool;
      Reset : Bool;
   END_VAR
   VAR_OUTPUT
      "Entry Conveyor" : Bool;
      "Load Conveyor" : Bool;
      "Target Position" : DInt;
      "P1 Step" : Bool;
      "P2 Step" : Bool;
      "P3 Step" : Bool;
      "P4 Step" : Bool;
      "P5 Step" : Bool;
      "P6 Step" : Bool;
      "Forks Left" : Bool;
      "Forks Right" : Bool;
      "Crane Lift" : Bool;
      "P3 Positive Edge Memory" : Bool;
   END_VAR
   VAR
      IEC_Timer_0_Instance : TON_TIME;
      IEC_Timer_0_Instance_1 : TON_TIME;
      IEC_Timer_0_Instance_2 : TON_TIME;
   END_VAR
   VAR RETAIN
      IEC_Counter_0_Instance : CTU_INT;
   END_VAR
   VAR
      IEC_Timer_0_Instance_3 : TON_TIME;
      IEC_Timer_0_Instance_4 : TON_TIME;
      IEC_Timer_0_Instance_5 : TON_TIME;
      IEC_Timer_0_Instance_6 : TON_TIME;
   END_VAR
   VAR_TEMP   // added for the SCL form of the ladder/FBD networks
      _w1 : Bool;
   END_VAR
BEGIN

REGION Network 1: Entry Conveyor
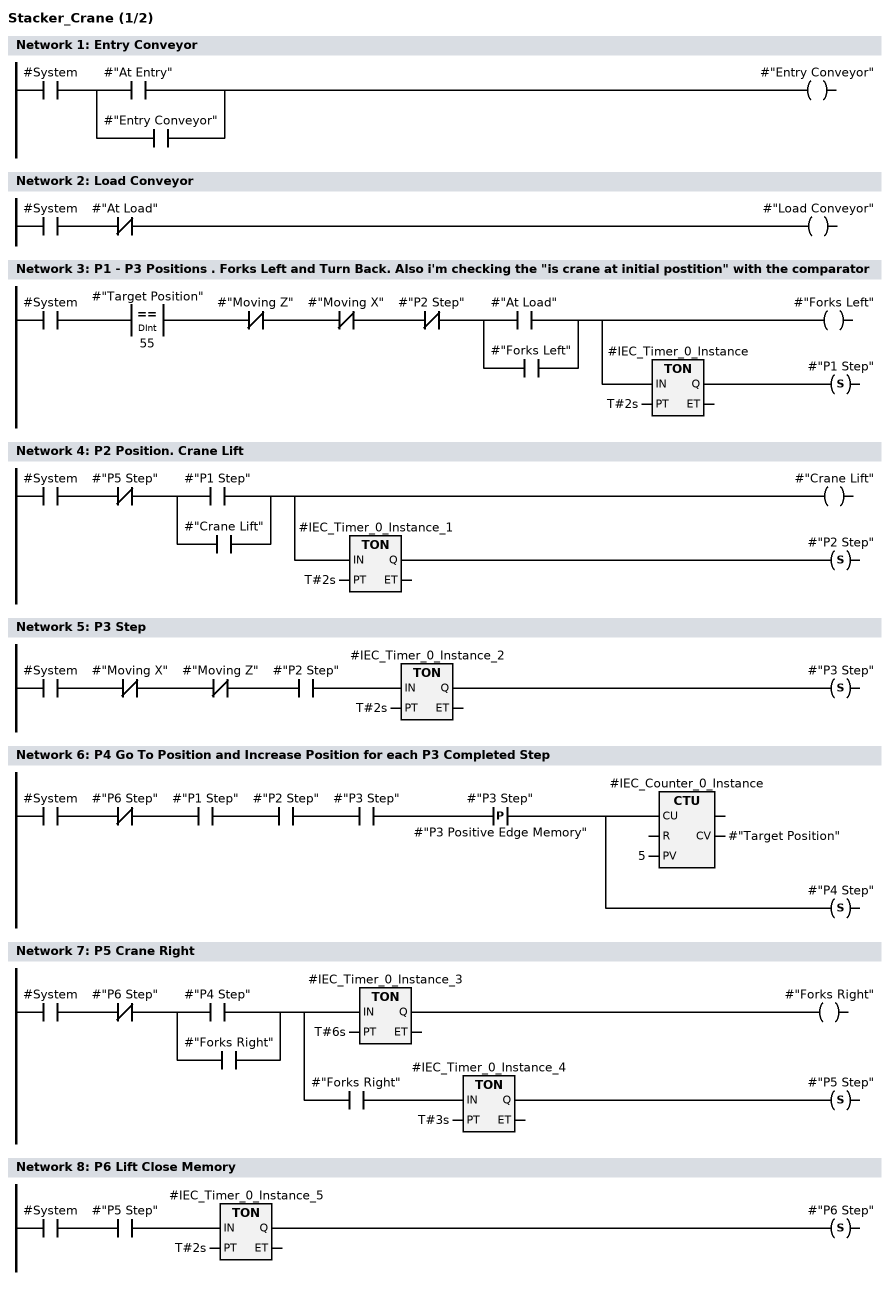
   RUNG wire#powerrail
      Contact( #System )
      wire#w1
      Contact( #"At Entry" )
      wire#w2
      Coil( #"Entry Conveyor" )
   END_RUNG
   RUNG wire#w1
      Contact( #"Entry Conveyor" )
   END_RUNG wire#w2
   // the same network as SCL:
   #"Entry Conveyor" := #System AND (#"At Entry" OR #"Entry Conveyor");
END_REGION

REGION Network 2: Load Conveyor
   RUNG wire#powerrail
      Contact( #System )
      I_Contact( #"At Load" )
      Coil( #"Load Conveyor" )
   END_RUNG
   // the same network as SCL:
   #"Load Conveyor" := #System AND NOT #"At Load";
END_REGION

REGION Network 3: P1 - P3 Positions . Forks Left and Turn Back. Also i'm checking the "is crane at initial postition" with the comparator
   #"Forks Left" := #System AND (#"Target Position" = 55) AND NOT #"Moving Z" AND NOT #"Moving X" AND NOT #"P2 Step" AND (#"At Load" OR #"Forks Left");
   #IEC_Timer_0_Instance(IN := #"Forks Left", PT := T#2s);   // TON
   IF #IEC_Timer_0_Instance.Q THEN #"P1 Step" := TRUE; END_IF;
END_REGION

REGION Network 4: P2 Position. Crane Lift
   #"Crane Lift" := #System AND NOT #"P5 Step" AND (#"P1 Step" OR #"Crane Lift");
   #IEC_Timer_0_Instance_1(IN := #"Crane Lift", PT := T#2s);   // TON
   IF #IEC_Timer_0_Instance_1.Q THEN #"P2 Step" := TRUE; END_IF;
END_REGION

REGION Network 5: P3 Step
   #IEC_Timer_0_Instance_2(IN := #System AND NOT #"Moving X" AND NOT #"Moving Z" AND #"P2 Step", PT := T#2s);   // TON
   IF #IEC_Timer_0_Instance_2.Q THEN #"P3 Step" := TRUE; END_IF;
END_REGION

REGION Network 6: P4 Go To Position and Increase Position for each P3 Completed Step
   #_w1 := #System AND NOT #"P6 Step" AND #"P1 Step" AND #"P2 Step" AND #"P3 Step" AND #"P3 Step" AND NOT #"P3 Positive Edge Memory";   // rising edge of #"P3 Step"
   #"P3 Positive Edge Memory" := #"P3 Step";
   #IEC_Counter_0_Instance(CU := #_w1, PV := 5, CV => #"Target Position");   // CTU
   IF #_w1 THEN #"P4 Step" := TRUE; END_IF;
END_REGION

REGION Network 7: P5 Crane Right
   #_w1 := #System AND NOT #"P6 Step" AND (#"P4 Step" OR #"Forks Right");
   #IEC_Timer_0_Instance_3(IN := #_w1, PT := T#6s);   // TON
   #"Forks Right" := #IEC_Timer_0_Instance_3.Q;
   #IEC_Timer_0_Instance_4(IN := #_w1 AND #"Forks Right", PT := T#3s);   // TON
   IF #IEC_Timer_0_Instance_4.Q THEN #"P5 Step" := TRUE; END_IF;
END_REGION

REGION Network 8: P6 Lift Close Memory
   #IEC_Timer_0_Instance_5(IN := #System AND #"P5 Step", PT := T#2s);   // TON
   IF #IEC_Timer_0_Instance_5.Q THEN #"P6 Step" := TRUE; END_IF;
END_REGION

REGION Network 9: Crane initial position
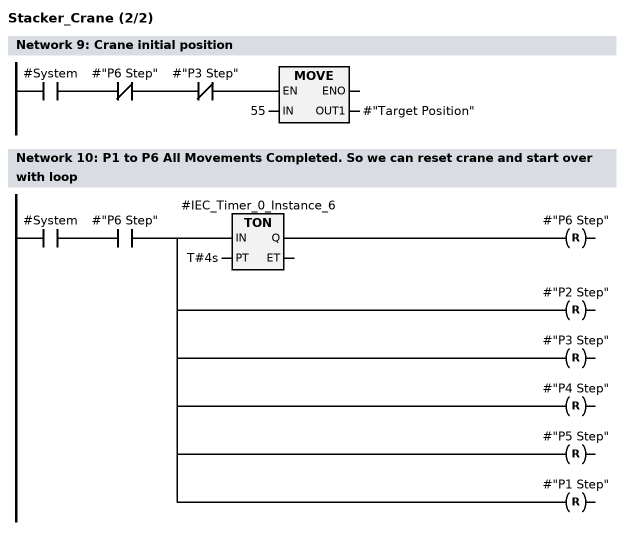
   RUNG wire#powerrail
      Contact( #System )
      I_Contact( #"P6 Step" )
      I_Contact( #"P3 Step" )
      Move(in := 55, out1 => #"Target Position")
   END_RUNG
   // the same network as SCL:
   IF #System AND NOT #"P6 Step" AND NOT #"P3 Step" THEN #"Target Position" := 55; END_IF;
END_REGION

REGION Network 10: P1 to P6 All Movements Completed. So we can reset crane and start over with loop
   #_w1 := #System AND #"P6 Step";
   #IEC_Timer_0_Instance_6(IN := #_w1, PT := T#4s);   // TON
   IF #IEC_Timer_0_Instance_6.Q THEN #"P6 Step" := FALSE; END_IF;
   IF #_w1 THEN
       #"P2 Step" := FALSE;
       #"P3 Step" := FALSE;
       #"P4 Step" := FALSE;
       #"P5 Step" := FALSE;
       #"P1 Step" := FALSE;
   END_IF;
END_REGION
END_FUNCTION_BLOCK

FUNCTION_BLOCK "Turn Table Right"   // FB5, LAD
{ S7_Optimized_Access := 'TRUE' }
VERSION : 0.1
   VAR_INPUT
      system : Bool;
      "Elevator Completed" : Bool;
      "Turn Table Front Limit" : Bool;
      "Turn Table Limit 0" : Bool;
      "Turn Table Limit 90" : Bool;
   END_VAR
   VAR_OUTPUT
      "Turn Table Input Roll" : Bool;
      "Turn Table Exit Roll" : Bool;
      "Turn Table Turn" : Bool;
      "Turn Table Completed" : Bool;
      "Turn Table is Busy" : Bool;
   END_VAR
   VAR
      IEC_Timer_0_Instance : TON_TIME;
   END_VAR
   VAR_TEMP   // added for the SCL form of the ladder/FBD networks
      _w1 : Bool;
   END_VAR
BEGIN

REGION Network 1: start turn table roll when elevator movements completed. and stop it when front limit sensor triggered
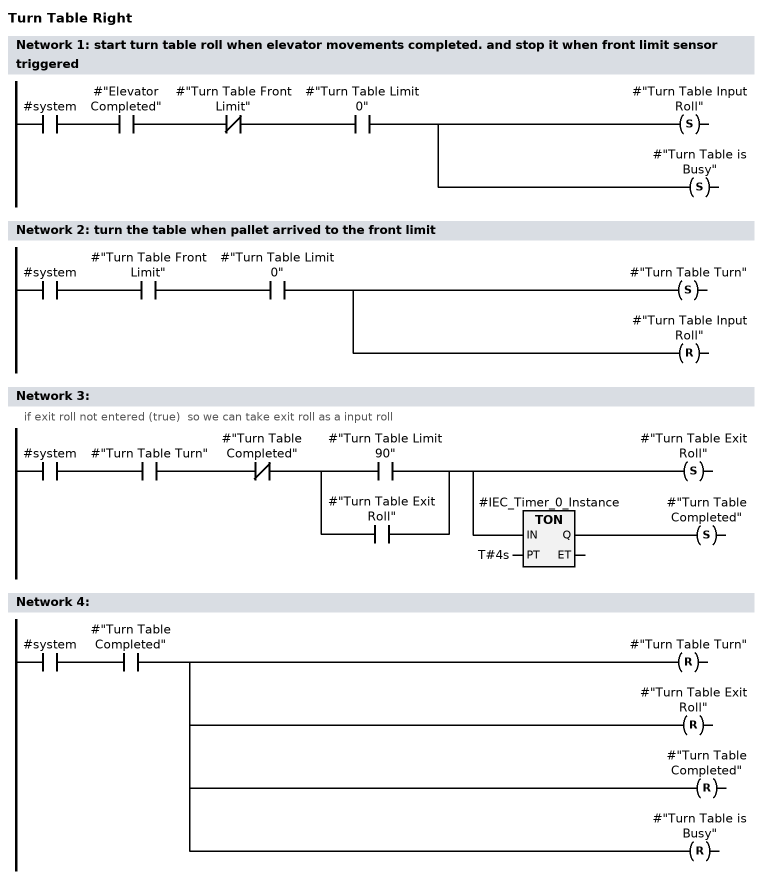
   RUNG wire#powerrail
      Contact( #system )
      Contact( #"Elevator Completed" )
      I_Contact( #"Turn Table Front Limit" )
      Contact( #"Turn Table Limit 0" )
      wire#w1
      S_Coil( #"Turn Table Input Roll" )
   END_RUNG
   RUNG wire#w1
      S_Coil( #"Turn Table is Busy" )
   END_RUNG
   // the same network as SCL:
   IF #system AND #"Elevator Completed" AND NOT #"Turn Table Front Limit" AND #"Turn Table Limit 0" THEN
       #"Turn Table Input Roll" := TRUE;
       #"Turn Table is Busy" := TRUE;
   END_IF;
END_REGION

REGION Network 2: turn the table when pallet arrived to the front limit
   RUNG wire#powerrail
      Contact( #system )
      Contact( #"Turn Table Front Limit" )
      Contact( #"Turn Table Limit 0" )
      wire#w1
      S_Coil( #"Turn Table Turn" )
   END_RUNG
   RUNG wire#w1
      R_Coil( #"Turn Table Input Roll" )
   END_RUNG
   // the same network as SCL:
   IF #system AND #"Turn Table Front Limit" AND #"Turn Table Limit 0" THEN
       #"Turn Table Turn" := TRUE;
       #"Turn Table Input Roll" := FALSE;
   END_IF;
END_REGION

REGION Network 3
   // if exit roll not entered (true)  so we can take exit roll as a input roll
   #_w1 := #system AND #"Turn Table Turn" AND NOT #"Turn Table Completed" AND (#"Turn Table Limit 90" OR #"Turn Table Exit Roll");
   IF #_w1 THEN #"Turn Table Exit Roll" := TRUE; END_IF;
   #IEC_Timer_0_Instance(IN := #_w1, PT := T#4s);   // TON
   IF #IEC_Timer_0_Instance.Q THEN #"Turn Table Completed" := TRUE; END_IF;
END_REGION

REGION Network 4
   RUNG wire#powerrail
      Contact( #system )
      Contact( #"Turn Table Completed" )
      wire#w1
      R_Coil( #"Turn Table Turn" )
   END_RUNG
   RUNG wire#w1
      R_Coil( #"Turn Table Exit Roll" )
   END_RUNG
   RUNG wire#w1
      R_Coil( #"Turn Table Completed" )
   END_RUNG
   RUNG wire#w1
      R_Coil( #"Turn Table is Busy" )
   END_RUNG
   // the same network as SCL:
   IF #system AND #"Turn Table Completed" THEN
       #"Turn Table Turn" := FALSE;
       #"Turn Table Exit Roll" := FALSE;
   END_IF;
   #_w1 := #system AND #"Turn Table Completed";
   IF #_w1 THEN
       #"Turn Table Completed" := FALSE;
       #"Turn Table is Busy" := FALSE;
   END_IF;
END_REGION
END_FUNCTION_BLOCK

FUNCTION_BLOCK "Palletizer"   // FB6, LAD
{ S7_Optimized_Access := 'TRUE' }
VERSION : 0.1
   VAR
      IEC_Timer_0_Instance : TON_TIME;
      IEC_Timer_0_Instance_1 : TON_TIME;
      IEC_Timer_0_Instance_2 : TON_TIME;
   END_VAR
   VAR RETAIN
      IEC_Counter_0_Instance : CTU_INT;
   END_VAR
   VAR_TEMP   // added for the SCL form of the ladder/FBD networks
      _w1 : Bool;
   END_VAR
BEGIN

REGION Network 1: Open Belt + all time
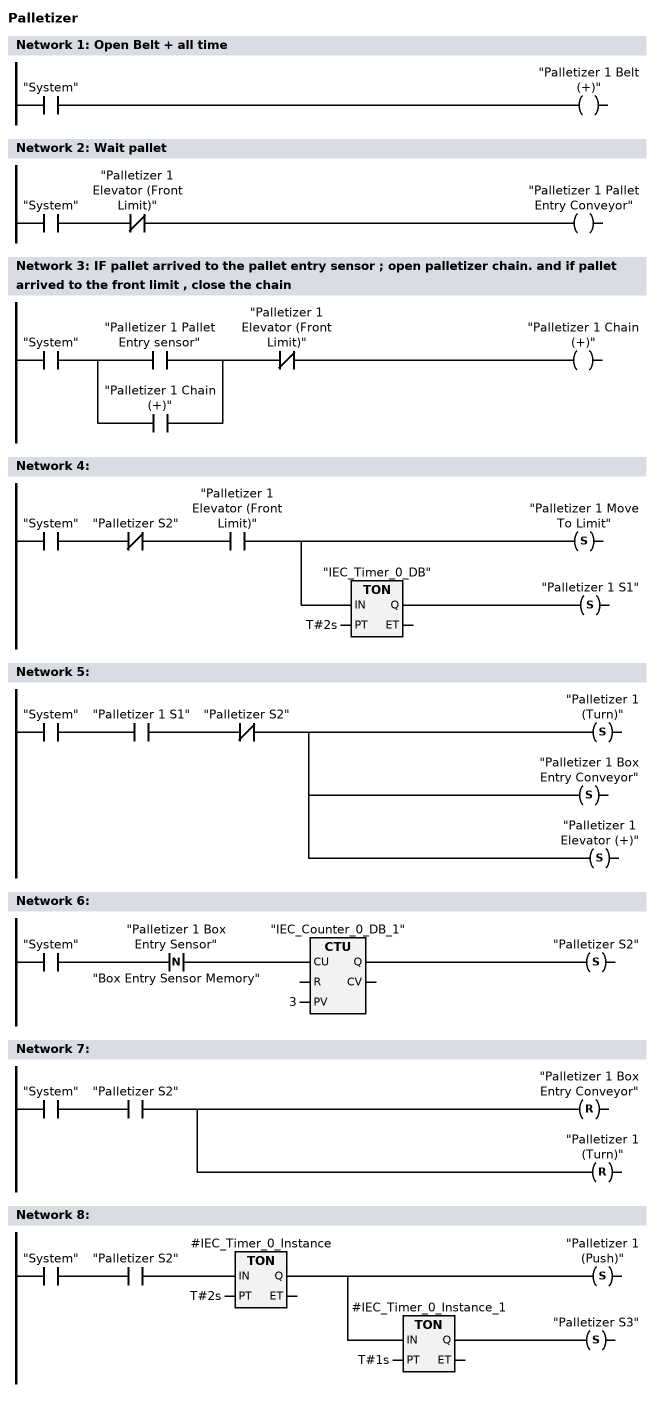
   RUNG wire#powerrail
      Contact( "System" )
      Coil( "Palletizer 1 Belt (+)" )
   END_RUNG
   // the same network as SCL:
   "Palletizer 1 Belt (+)" := "System";
END_REGION

REGION Network 2: Wait pallet
   RUNG wire#powerrail
      Contact( "System" )
      I_Contact( "Palletizer 1 Elevator (Front Limit)" )
      Coil( "Palletizer 1 Pallet Entry Conveyor" )
   END_RUNG
   // the same network as SCL:
   "Palletizer 1 Pallet Entry Conveyor" := "System" AND NOT "Palletizer 1 Elevator (Front Limit)";
END_REGION

REGION Network 3: IF pallet arrived to the pallet entry sensor ; open palletizer chain. and if pallet arrived to the front limit , close the chain
   RUNG wire#powerrail
      Contact( "System" )
      wire#w1
      Contact( "Palletizer 1 Pallet Entry sensor" )
      wire#w2
      I_Contact( "Palletizer 1 Elevator (Front Limit)" )
      Coil( "Palletizer 1 Chain (+)" )
   END_RUNG
   RUNG wire#w1
      Contact( "Palletizer 1 Chain (+)" )
   END_RUNG wire#w2
   // the same network as SCL:
   "Palletizer 1 Chain (+)" := "System" AND ("Palletizer 1 Pallet Entry sensor" OR "Palletizer 1 Chain (+)") AND NOT "Palletizer 1 Elevator (Front Limit)";
END_REGION

REGION Network 4
   #_w1 := "System" AND NOT "Palletizer S2" AND "Palletizer 1 Elevator (Front Limit)";
   IF #_w1 THEN "Palletizer 1 Move To Limit" := TRUE; END_IF;
   "IEC_Timer_0_DB".TON(IN := #_w1, PT := T#2s);
   IF "IEC_Timer_0_DB".Q THEN "Palletizer 1 S1" := TRUE; END_IF;
END_REGION

REGION Network 5
   RUNG wire#powerrail
      Contact( "System" )
      Contact( "Palletizer 1 S1" )
      I_Contact( "Palletizer S2" )
      wire#w1
      S_Coil( "Palletizer 1 (Turn)" )
   END_RUNG
   RUNG wire#w1
      S_Coil( "Palletizer 1 Box Entry Conveyor" )
   END_RUNG
   RUNG wire#w1
      S_Coil( "Palletizer 1 Elevator (+)" )
   END_RUNG
   // the same network as SCL:
   IF "System" AND "Palletizer 1 S1" AND NOT "Palletizer S2" THEN
       "Palletizer 1 (Turn)" := TRUE;
       "Palletizer 1 Box Entry Conveyor" := TRUE;
       "Palletizer 1 Elevator (+)" := TRUE;
   END_IF;
END_REGION

REGION Network 6
   #_w1 := "System" AND NOT "Palletizer 1 Box Entry Sensor" AND "Box Entry Sensor Memory";   // falling edge of "Palletizer 1 Box Entry Sensor"
   "Box Entry Sensor Memory" := "Palletizer 1 Box Entry Sensor";
   "IEC_Counter_0_DB_1".CTU(CU := #_w1, PV := 3);
   IF "IEC_Counter_0_DB_1".Q THEN "Palletizer S2" := TRUE; END_IF;
END_REGION

REGION Network 7
   RUNG wire#powerrail
      Contact( "System" )
      Contact( "Palletizer S2" )
      wire#w1
      R_Coil( "Palletizer 1 Box Entry Conveyor" )
   END_RUNG
   RUNG wire#w1
      R_Coil( "Palletizer 1 (Turn)" )
   END_RUNG
   // the same network as SCL:
   IF "System" AND "Palletizer S2" THEN
       "Palletizer 1 Box Entry Conveyor" := FALSE;
       "Palletizer 1 (Turn)" := FALSE;
   END_IF;
END_REGION

REGION Network 8
   #IEC_Timer_0_Instance(IN := "System" AND "Palletizer S2", PT := T#2s);   // TON
   IF #IEC_Timer_0_Instance.Q THEN "Palletizer 1 (Push)" := TRUE; END_IF;
   #IEC_Timer_0_Instance_1(IN := #IEC_Timer_0_Instance.Q, PT := T#1s);   // TON
   IF #IEC_Timer_0_Instance_1.Q THEN "Palletizer S3" := TRUE; END_IF;
END_REGION
END_FUNCTION_BLOCK

FUNCTION "MHJ-PLC-Lab-Function-S71200" : Void   // FC9000, SCL
{ S7_Optimized_Access := 'TRUE' }
VERSION : 0.1
   VAR_TEMP
      rdTimeReturn : Int;
      outputTime : DTL;
      SyncVal : Byte;
      forVal : Int;
      forVal_2 : Int;
      Value : Byte;
   END_VAR
   VAR CONSTANT
      CompVal : Byte := 16#34;
      Value_01 : Byte := 16#11;
      Value_01_DW : DWord := 16#A165_D992;
      Value_02_DW : DWord := 16#58BE_4401;
   END_VAR
BEGIN

   #Value:=PEEK(area := 16#82,
        dbNumber := 0,
        byteOffset := 511);
   #Value := #Value + 1;

   POKE(area := 16#82,
        dbNumber := 0,
        byteOffset := 511,
        value := #Value);

   POKE(area:=16#81,
        dbNumber:=0,
        byteOffset:=1016,
        value:=#Value_01_DW);
   POKE(area := 16#81,
        dbNumber := 0,
        byteOffset := 1020,
        value := #Value_02_DW);

   POKE(area := 16#81,
        dbNumber := 0,
        byteOffset := 511,
        value := B#16#00);

   FOR #forVal := 0 TO 120 DO
       FOR #forVal_2:=0 TO 10 DO
           #rdTimeReturn:=RD_SYS_T(#outputTime);
           #rdTimeReturn := WR_SYS_T(#outputTime);
           #rdTimeReturn := RD_SYS_T(#outputTime);
           #rdTimeReturn := WR_SYS_T(#outputTime);
       END_FOR;
       #SyncVal:= PEEK(area := 16#81,
                      dbNumber := 0,
                      byteOffset := 511);
       IF #SyncVal = #CompVal THEN
          GOTO M_1;
       END_IF;
   END_FOR;
   RETURN;

   M_1:
   POKE(area := 16#81,
        dbNumber := 0,
        byteOffset := 511,
        value := B#16#0);
END_FUNCTION

ORGANIZATION_BLOCK "Main"   // OB1, LAD, ProgramCycle
TITLE = "Main Program Sweep (Cycle)"
{ S7_Optimized_Access := 'TRUE' }
VERSION : 0.1
   VAR_INPUT
      Initial_Call : Bool;   // Initial call of this OB
      Remanence : Bool;   // =True, if remanent data are available
   END_VAR
BEGIN

REGION Network 1
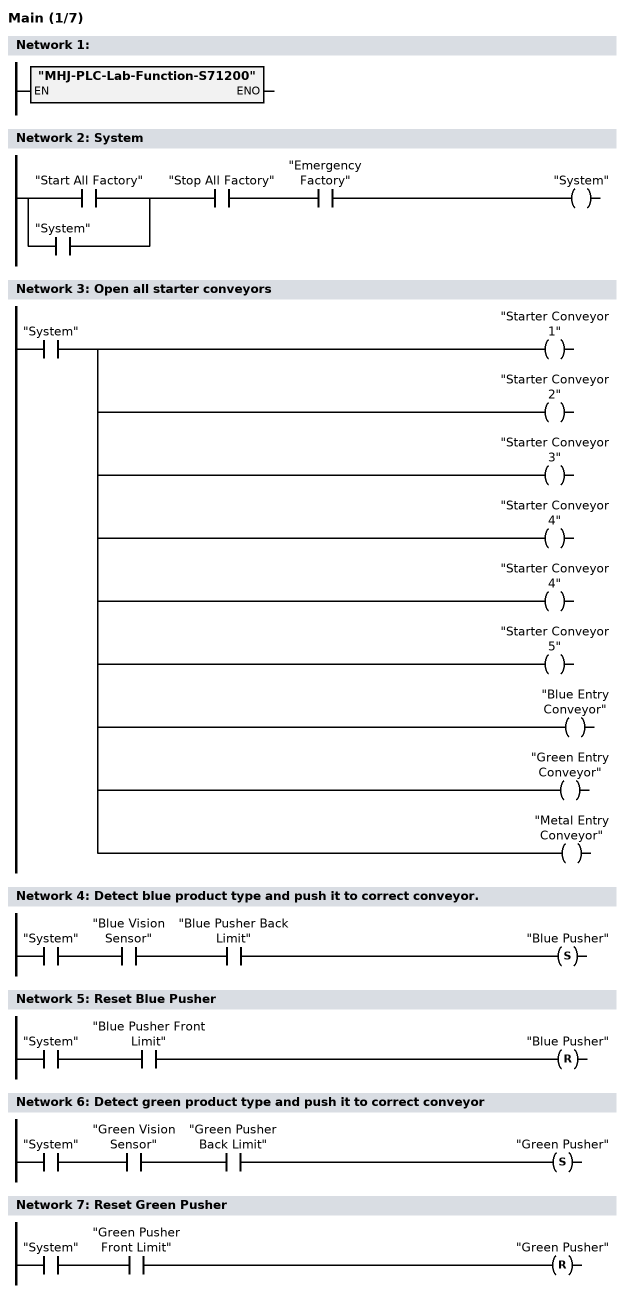
   RUNG wire#powerrail
      "MHJ-PLC-Lab-Function-S71200"()
   END_RUNG
   // the same network as SCL:
   "MHJ-PLC-Lab-Function-S71200"();
END_REGION

REGION Network 2: System
   RUNG wire#powerrail
      Contact( "Start All Factory" )
      wire#w1
      Contact( "Stop All Factory" )
      Contact( "Emergency Factory" )
      Coil( "System" )
   END_RUNG
   RUNG wire#powerrail
      Contact( "System" )
   END_RUNG wire#w1
   // the same network as SCL:
   "System" := ("Start All Factory" OR "System") AND "Stop All Factory" AND "Emergency Factory";
END_REGION

REGION Network 3: Open all starter conveyors
   RUNG wire#powerrail
      Contact( "System" )
      wire#w1
      Coil( "Starter Conveyor 1" )
   END_RUNG
   RUNG wire#w1
      Coil( "Starter Conveyor 2" )
   END_RUNG
   RUNG wire#w1
      Coil( "Starter Conveyor 3" )
   END_RUNG
   RUNG wire#w1
      Coil( "Starter Conveyor 4" )
   END_RUNG
   RUNG wire#w1
      Coil( "Starter Conveyor 4" )
   END_RUNG
   RUNG wire#w1
      Coil( "Starter Conveyor 5" )
   END_RUNG
   RUNG wire#w1
      Coil( "Blue Entry Conveyor" )
   END_RUNG
   RUNG wire#w1
      Coil( "Green Entry Conveyor" )
   END_RUNG
   RUNG wire#w1
      Coil( "Metal Entry Conveyor" )
   END_RUNG
   // the same network as SCL:
   "Starter Conveyor 1" := "System";
   "Starter Conveyor 2" := "System";
   "Starter Conveyor 3" := "System";
   "Starter Conveyor 4" := "System";
   "Starter Conveyor 4" := "System";
   "Starter Conveyor 5" := "System";
   "Blue Entry Conveyor" := "System";
   "Green Entry Conveyor" := "System";
   "Metal Entry Conveyor" := "System";
END_REGION

REGION Network 4: Detect blue product type and push it to correct conveyor.
   RUNG wire#powerrail
      Contact( "System" )
      Contact( "Blue Vision Sensor" )
      Contact( "Blue Pusher Back Limit" )
      S_Coil( "Blue Pusher" )
   END_RUNG
   // the same network as SCL:
   IF "System" AND "Blue Vision Sensor" AND "Blue Pusher Back Limit" THEN "Blue Pusher" := TRUE; END_IF;
END_REGION

REGION Network 5: Reset Blue Pusher
   RUNG wire#powerrail
      Contact( "System" )
      Contact( "Blue Pusher Front Limit" )
      R_Coil( "Blue Pusher" )
   END_RUNG
   // the same network as SCL:
   IF "System" AND "Blue Pusher Front Limit" THEN "Blue Pusher" := FALSE; END_IF;
END_REGION

REGION Network 6: Detect green product type and push it to correct conveyor
   RUNG wire#powerrail
      Contact( "System" )
      Contact( "Green Vision Sensor" )
      Contact( "Green Pusher Back Limit" )
      S_Coil( "Green Pusher" )
   END_RUNG
   // the same network as SCL:
   IF "System" AND "Green Vision Sensor" AND "Green Pusher Back Limit" THEN "Green Pusher" := TRUE; END_IF;
END_REGION

REGION Network 7: Reset Green Pusher
   RUNG wire#powerrail
      Contact( "System" )
      Contact( "Green Pusher Front Limit" )
      R_Coil( "Green Pusher" )
   END_RUNG
   // the same network as SCL:
   IF "System" AND "Green Pusher Front Limit" THEN "Green Pusher" := FALSE; END_IF;
END_REGION

REGION Network 8: Detect metal product type and push it to correct conveyor
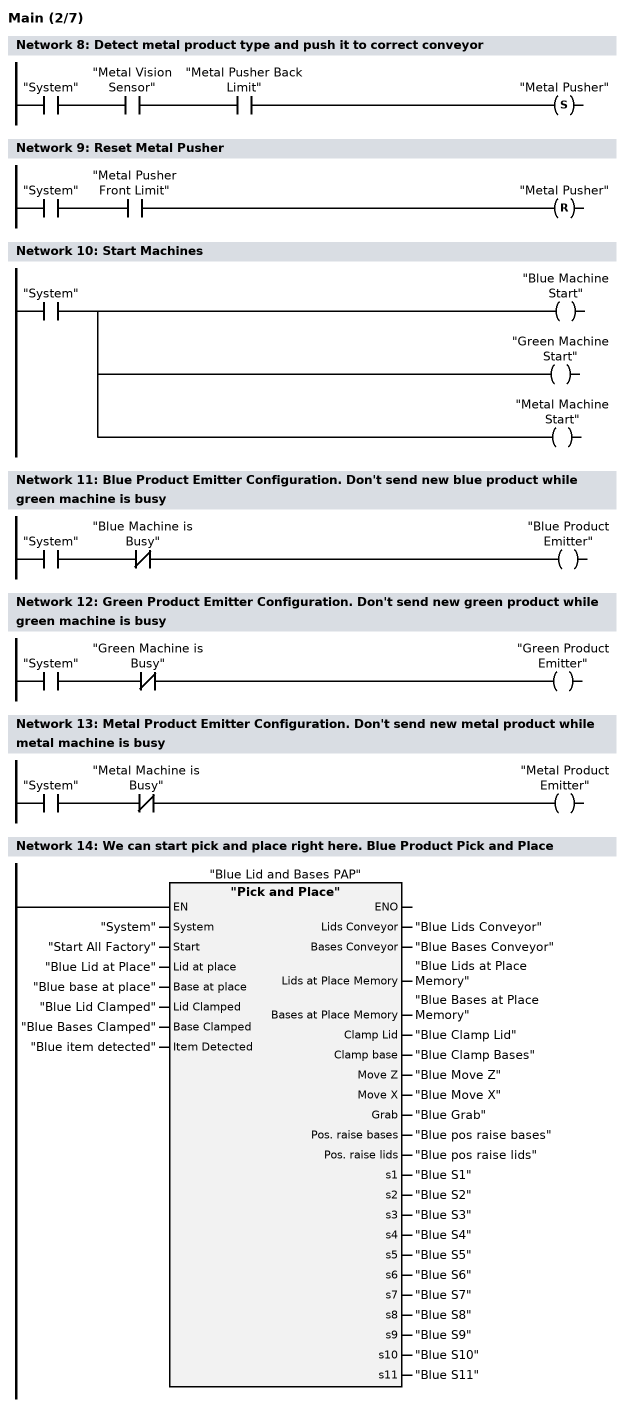
   RUNG wire#powerrail
      Contact( "System" )
      Contact( "Metal Vision Sensor" )
      Contact( "Metal Pusher Back Limit" )
      S_Coil( "Metal Pusher" )
   END_RUNG
   // the same network as SCL:
   IF "System" AND "Metal Vision Sensor" AND "Metal Pusher Back Limit" THEN "Metal Pusher" := TRUE; END_IF;
END_REGION

REGION Network 9: Reset Metal Pusher
   RUNG wire#powerrail
      Contact( "System" )
      Contact( "Metal Pusher Front Limit" )
      R_Coil( "Metal Pusher" )
   END_RUNG
   // the same network as SCL:
   IF "System" AND "Metal Pusher Front Limit" THEN "Metal Pusher" := FALSE; END_IF;
END_REGION

REGION Network 10: Start Machines
   RUNG wire#powerrail
      Contact( "System" )
      wire#w1
      Coil( "Blue Machine Start" )
   END_RUNG
   RUNG wire#w1
      Coil( "Green Machine Start" )
   END_RUNG
   RUNG wire#w1
      Coil( "Metal Machine Start" )
   END_RUNG
   // the same network as SCL:
   "Blue Machine Start" := "System";
   "Green Machine Start" := "System";
   "Metal Machine Start" := "System";
END_REGION

REGION Network 11: Blue Product Emitter Configuration. Don't send new blue product while green machine is busy
   RUNG wire#powerrail
      Contact( "System" )
      I_Contact( "Blue Machine is Busy" )
      Coil( "Blue Product Emitter" )
   END_RUNG
   // the same network as SCL:
   "Blue Product Emitter" := "System" AND NOT "Blue Machine is Busy";
END_REGION

REGION Network 12: Green Product Emitter Configuration. Don't send new green product while green machine is busy
   RUNG wire#powerrail
      Contact( "System" )
      I_Contact( "Green Machine is Busy" )
      Coil( "Green Product Emitter" )
   END_RUNG
   // the same network as SCL:
   "Green Product Emitter" := "System" AND NOT "Green Machine is Busy";
END_REGION

REGION Network 13: Metal Product Emitter Configuration. Don't send new metal product while metal machine is busy
   RUNG wire#powerrail
      Contact( "System" )
      I_Contact( "Metal Machine is Busy" )
      Coil( "Metal Product Emitter" )
   END_RUNG
   // the same network as SCL:
   "Metal Product Emitter" := "System" AND NOT "Metal Machine is Busy";
END_REGION

REGION Network 14: We can start pick and place right here. Blue Product Pick and Place
   RUNG wire#powerrail
      "Blue Lid and Bases PAP"(System := "System", Start := "Start All Factory", "Lid at place" := "Blue Lid at Place", "Base at place" := "Blue base at place", "Lid Clamped" := "Blue Lid Clamped", "Base Clamped" := "Blue Bases Clamped", "Item Detected" := "Blue item detected", "Lids Conveyor" => "Blue Lids Conveyor", "Bases Conveyor" => "Blue Bases Conveyor", "Lids at Place Memory" => "Blue Lids at Place Memory", "Bases at Place Memory" => "Blue Bases at Place Memory", "Clamp Lid" => "Blue Clamp Lid", "Clamp base" => "Blue Clamp Bases", "Move Z" => "Blue Move Z", "Move X" => "Blue Move X", Grab => "Blue Grab", "Pos. raise bases" => "Blue pos raise bases", "Pos. raise lids" => "Blue pos raise lids", s1 => "Blue S1", s2 => "Blue S2", s3 => "Blue S3", s4 => "Blue S4", s5 => "Blue S5", s6 => "Blue S6", s7 => "Blue S7", s8 => "Blue S8", s9 => "Blue S9", s10 => "Blue S10", s11 => "Blue S11")
   END_RUNG
   // the same network as SCL:
   "Blue Lid and Bases PAP"(System := "System",   // "Pick and Place"
                           Start := "Start All Factory",
                           "Lid at place" := "Blue Lid at Place",
                           "Base at place" := "Blue base at place",
                           "Lid Clamped" := "Blue Lid Clamped",
                           "Base Clamped" := "Blue Bases Clamped",
                           "Item Detected" := "Blue item detected",
                           "Lids Conveyor" => "Blue Lids Conveyor",
                           "Bases Conveyor" => "Blue Bases Conveyor",
                           "Lids at Place Memory" => "Blue Lids at Place Memory",
                           "Bases at Place Memory" => "Blue Bases at Place Memory",
                           "Clamp Lid" => "Blue Clamp Lid",
                           "Clamp base" => "Blue Clamp Bases",
                           "Move Z" => "Blue Move Z",
                           "Move X" => "Blue Move X",
                           Grab => "Blue Grab",
                           "Pos. raise bases" => "Blue pos raise bases",
                           "Pos. raise lids" => "Blue pos raise lids",
                           s1 => "Blue S1",
                           s2 => "Blue S2",
                           s3 => "Blue S3",
                           s4 => "Blue S4",
                           s5 => "Blue S5",
                           s6 => "Blue S6",
                           s7 => "Blue S7",
                           s8 => "Blue S8",
                           s9 => "Blue S9",
                           s10 => "Blue S10",
                           s11 => "Blue S11");
END_REGION

REGION Network 15: Green Product Pick and Place
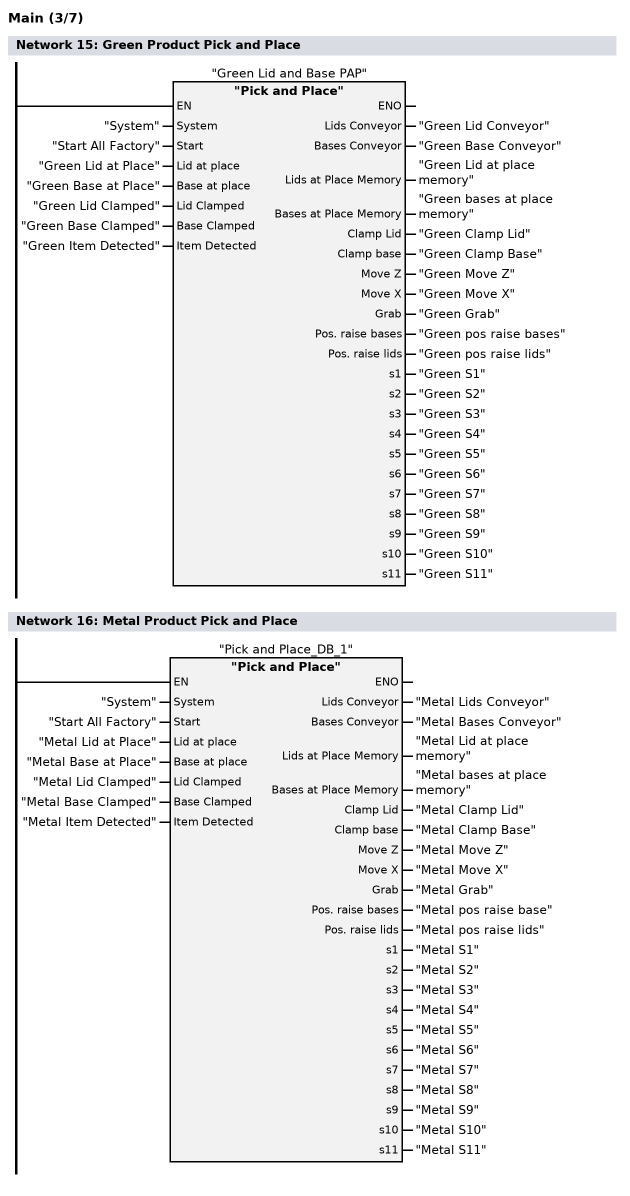
   RUNG wire#powerrail
      "Green Lid and Base PAP"(System := "System", Start := "Start All Factory", "Lid at place" := "Green Lid at Place", "Base at place" := "Green Base at Place", "Lid Clamped" := "Green Lid Clamped", "Base Clamped" := "Green Base Clamped", "Item Detected" := "Green Item Detected", "Lids Conveyor" => "Green Lid Conveyor", "Bases Conveyor" => "Green Base Conveyor", "Lids at Place Memory" => "Green Lid at place memory", "Bases at Place Memory" => "Green bases at place memory", "Clamp Lid" => "Green Clamp Lid", "Clamp base" => "Green Clamp Base", "Move Z" => "Green Move Z", "Move X" => "Green Move X", Grab => "Green Grab", "Pos. raise bases" => "Green pos raise bases", "Pos. raise lids" => "Green pos raise lids", s1 => "Green S1", s2 => "Green S2", s3 => "Green S3", s4 => "Green S4", s5 => "Green S5", s6 => "Green S6", s7 => "Green S7", s8 => "Green S8", s9 => "Green S9", s10 => "Green S10", s11 => "Green S11")
   END_RUNG
   // the same network as SCL:
   "Green Lid and Base PAP"(System := "System",   // "Pick and Place"
                           Start := "Start All Factory",
                           "Lid at place" := "Green Lid at Place",
                           "Base at place" := "Green Base at Place",
                           "Lid Clamped" := "Green Lid Clamped",
                           "Base Clamped" := "Green Base Clamped",
                           "Item Detected" := "Green Item Detected",
                           "Lids Conveyor" => "Green Lid Conveyor",
                           "Bases Conveyor" => "Green Base Conveyor",
                           "Lids at Place Memory" => "Green Lid at place memory",
                           "Bases at Place Memory" => "Green bases at place memory",
                           "Clamp Lid" => "Green Clamp Lid",
                           "Clamp base" => "Green Clamp Base",
                           "Move Z" => "Green Move Z",
                           "Move X" => "Green Move X",
                           Grab => "Green Grab",
                           "Pos. raise bases" => "Green pos raise bases",
                           "Pos. raise lids" => "Green pos raise lids",
                           s1 => "Green S1",
                           s2 => "Green S2",
                           s3 => "Green S3",
                           s4 => "Green S4",
                           s5 => "Green S5",
                           s6 => "Green S6",
                           s7 => "Green S7",
                           s8 => "Green S8",
                           s9 => "Green S9",
                           s10 => "Green S10",
                           s11 => "Green S11");
END_REGION

REGION Network 16: Metal Product Pick and Place
   RUNG wire#powerrail
      "Pick and Place_DB_1"(System := "System", Start := "Start All Factory", "Lid at place" := "Metal Lid at Place", "Base at place" := "Metal Base at Place", "Lid Clamped" := "Metal Lid Clamped", "Base Clamped" := "Metal Base Clamped", "Item Detected" := "Metal Item Detected", "Lids Conveyor" => "Metal Lids Conveyor", "Bases Conveyor" => "Metal Bases Conveyor", "Lids at Place Memory" => "Metal Lid at place memory", "Bases at Place Memory" => "Metal bases at place memory", "Clamp Lid" => "Metal Clamp Lid", "Clamp base" => "Metal Clamp Base", "Move Z" => "Metal Move Z", "Move X" => "Metal Move X", Grab => "Metal Grab", "Pos. raise bases" => "Metal pos raise base", "Pos. raise lids" => "Metal pos raise lids", s1 => "Metal S1", s2 => "Metal S2", s3 => "Metal S3", s4 => "Metal S4", s5 => "Metal S5", s6 => "Metal S6", s7 => "Metal S7", s8 => "Metal S8", s9 => "Metal S9", s10 => "Metal S10", s11 => "Metal S11")
   END_RUNG
   // the same network as SCL:
   "Pick and Place_DB_1"(System := "System",   // "Pick and Place"
                         Start := "Start All Factory",
                         "Lid at place" := "Metal Lid at Place",
                         "Base at place" := "Metal Base at Place",
                         "Lid Clamped" := "Metal Lid Clamped",
                         "Base Clamped" := "Metal Base Clamped",
                         "Item Detected" := "Metal Item Detected",
                         "Lids Conveyor" => "Metal Lids Conveyor",
                         "Bases Conveyor" => "Metal Bases Conveyor",
                         "Lids at Place Memory" => "Metal Lid at place memory",
                         "Bases at Place Memory" => "Metal bases at place memory",
                         "Clamp Lid" => "Metal Clamp Lid",
                         "Clamp base" => "Metal Clamp Base",
                         "Move Z" => "Metal Move Z",
                         "Move X" => "Metal Move X",
                         Grab => "Metal Grab",
                         "Pos. raise bases" => "Metal pos raise base",
                         "Pos. raise lids" => "Metal pos raise lids",
                         s1 => "Metal S1",
                         s2 => "Metal S2",
                         s3 => "Metal S3",
                         s4 => "Metal S4",
                         s5 => "Metal S5",
                         s6 => "Metal S6",
                         s7 => "Metal S7",
                         s8 => "Metal S8",
                         s9 => "Metal S9",
                         s10 => "Metal S10",
                         s11 => "Metal S11");
END_REGION

REGION Network 17: Blue Pallet Pick and Place
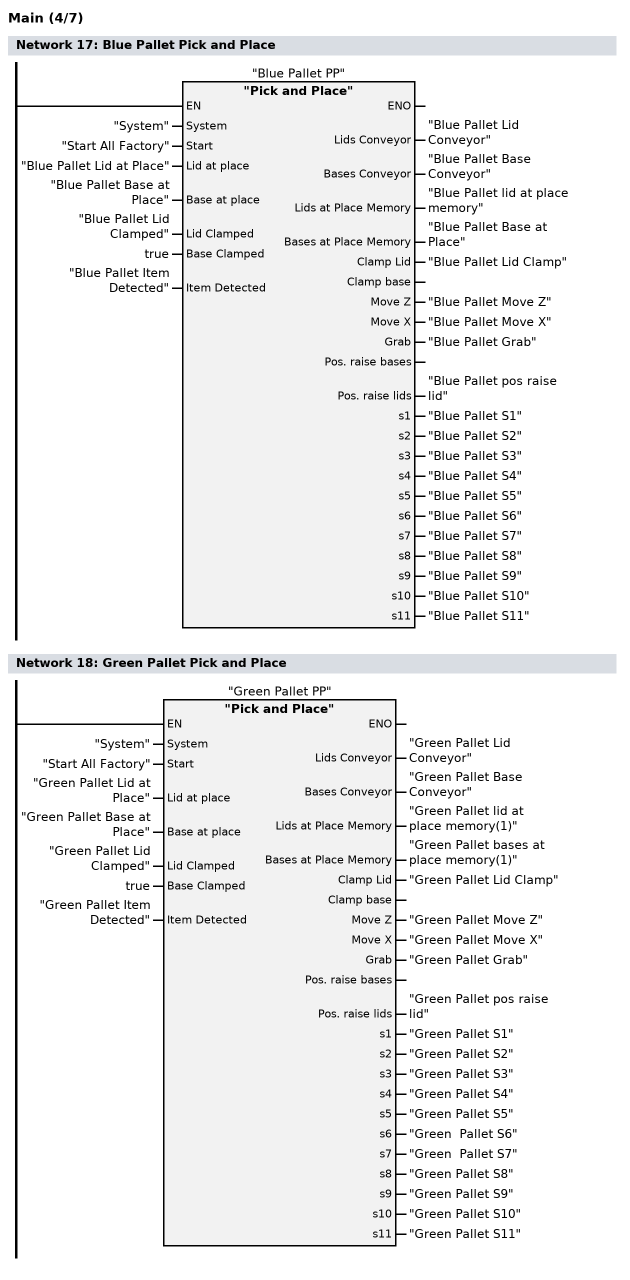
   RUNG wire#powerrail
      "Blue Pallet PP"(System := "System", Start := "Start All Factory", "Lid at place" := "Blue Pallet Lid at Place", "Base at place" := "Blue Pallet Base at Place", "Lid Clamped" := "Blue Pallet Lid Clamped", "Base Clamped" := true, "Item Detected" := "Blue Pallet Item Detected", "Lids Conveyor" => "Blue Pallet Lid Conveyor", "Bases Conveyor" => "Blue Pallet Base Conveyor", "Lids at Place Memory" => "Blue Pallet lid at place memory", "Bases at Place Memory" => "Blue Pallet Base at Place", "Clamp Lid" => "Blue Pallet Lid Clamp", "Clamp base" =>, "Move Z" => "Blue Pallet Move Z", "Move X" => "Blue Pallet Move X", Grab => "Blue Pallet Grab", "Pos. raise bases" =>, "Pos. raise lids" => "Blue Pallet pos raise lid", s1 => "Blue Pallet S1", s2 => "Blue Pallet S2", s3 => "Blue Pallet S3", s4 => "Blue Pallet S4", s5 => "Blue Pallet S5", s6 => "Blue Pallet S6", s7 => "Blue Pallet S7", s8 => "Blue Pallet S8", s9 => "Blue Pallet S9", s10 => "Blue Pallet S10", s11 => "Blue Pallet S11")
   END_RUNG
   // the same network as SCL:
   "Blue Pallet PP"(System := "System",   // "Pick and Place"
                    Start := "Start All Factory",
                    "Lid at place" := "Blue Pallet Lid at Place",
                    "Base at place" := "Blue Pallet Base at Place",
                    "Lid Clamped" := "Blue Pallet Lid Clamped",
                    "Base Clamped" := true,
                    "Item Detected" := "Blue Pallet Item Detected",
                    "Lids Conveyor" => "Blue Pallet Lid Conveyor",
                    "Bases Conveyor" => "Blue Pallet Base Conveyor",
                    "Lids at Place Memory" => "Blue Pallet lid at place memory",
                    "Bases at Place Memory" => "Blue Pallet Base at Place",
                    "Clamp Lid" => "Blue Pallet Lid Clamp",
                    "Move Z" => "Blue Pallet Move Z",
                    "Move X" => "Blue Pallet Move X",
                    Grab => "Blue Pallet Grab",
                    "Pos. raise lids" => "Blue Pallet pos raise lid",
                    s1 => "Blue Pallet S1",
                    s2 => "Blue Pallet S2",
                    s3 => "Blue Pallet S3",
                    s4 => "Blue Pallet S4",
                    s5 => "Blue Pallet S5",
                    s6 => "Blue Pallet S6",
                    s7 => "Blue Pallet S7",
                    s8 => "Blue Pallet S8",
                    s9 => "Blue Pallet S9",
                    s10 => "Blue Pallet S10",
                    s11 => "Blue Pallet S11");
END_REGION

REGION Network 18: Green Pallet Pick and Place
   RUNG wire#powerrail
      "Green Pallet PP"(System := "System", Start := "Start All Factory", "Lid at place" := "Green Pallet Lid at Place", "Base at place" := "Green Pallet Base at Place", "Lid Clamped" := "Green Pallet Lid Clamped", "Base Clamped" := true, "Item Detected" := "Green Pallet Item Detected", "Lids Conveyor" => "Green Pallet Lid Conveyor", "Bases Conveyor" => "Green Pallet Base Conveyor", "Lids at Place Memory" => "Green Pallet lid at place memory(1)", "Bases at Place Memory" => "Green Pallet bases at place memory(1)", "Clamp Lid" => "Green Pallet Lid Clamp", "Clamp base" =>, "Move Z" => "Green Pallet Move Z", "Move X" => "Green Pallet Move X", Grab => "Green Pallet Grab", "Pos. raise bases" =>, "Pos. raise lids" => "Green Pallet pos raise lid", s1 => "Green Pallet S1", s2 => "Green Pallet S2", s3 => "Green Pallet S3", s4 => "Green Pallet S4", s5 => "Green Pallet S5", s6 => "Green  Pallet S6", s7 => "Green  Pallet S7", s8 => "Green Pallet S8", s9 => "Green Pallet S9", s10 => "Green Pallet S10", s11 => "Green Pallet S11")
   END_RUNG
   // the same network as SCL:
   "Green Pallet PP"(System := "System",   // "Pick and Place"
                     Start := "Start All Factory",
                     "Lid at place" := "Green Pallet Lid at Place",
                     "Base at place" := "Green Pallet Base at Place",
                     "Lid Clamped" := "Green Pallet Lid Clamped",
                     "Base Clamped" := true,
                     "Item Detected" := "Green Pallet Item Detected",
                     "Lids Conveyor" => "Green Pallet Lid Conveyor",
                     "Bases Conveyor" => "Green Pallet Base Conveyor",
                     "Lids at Place Memory" => "Green Pallet lid at place memory(1)",
                     "Bases at Place Memory" => "Green Pallet bases at place memory(1)",
                     "Clamp Lid" => "Green Pallet Lid Clamp",
                     "Move Z" => "Green Pallet Move Z",
                     "Move X" => "Green Pallet Move X",
                     Grab => "Green Pallet Grab",
                     "Pos. raise lids" => "Green Pallet pos raise lid",
                     s1 => "Green Pallet S1",
                     s2 => "Green Pallet S2",
                     s3 => "Green Pallet S3",
                     s4 => "Green Pallet S4",
                     s5 => "Green Pallet S5",
                     s6 => "Green  Pallet S6",
                     s7 => "Green  Pallet S7",
                     s8 => "Green Pallet S8",
                     s9 => "Green Pallet S9",
                     s10 => "Green Pallet S10",
                     s11 => "Green Pallet S11");
END_REGION

REGION Network 19: Metal Pallet Pick and Place
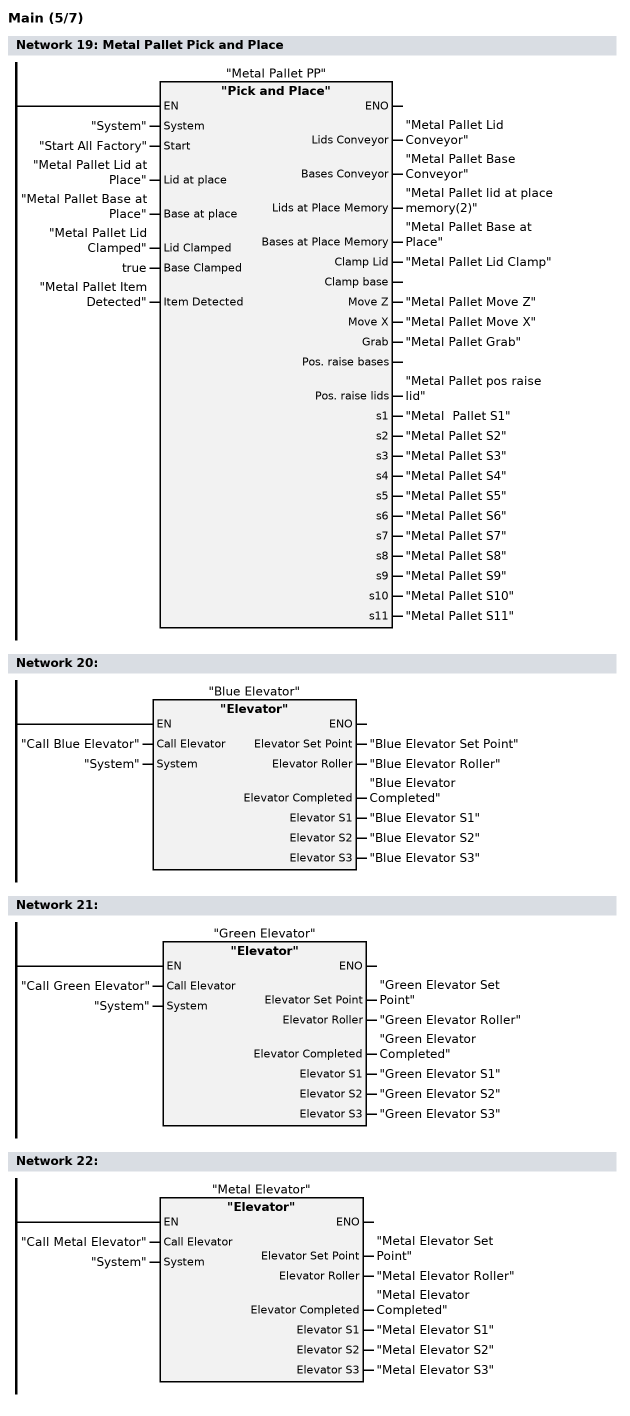
   RUNG wire#powerrail
      "Metal Pallet PP"(System := "System", Start := "Start All Factory", "Lid at place" := "Metal Pallet Lid at Place", "Base at place" := "Metal Pallet Base at Place", "Lid Clamped" := "Metal Pallet Lid Clamped", "Base Clamped" := true, "Item Detected" := "Metal Pallet Item Detected", "Lids Conveyor" => "Metal Pallet Lid Conveyor", "Bases Conveyor" => "Metal Pallet Base Conveyor", "Lids at Place Memory" => "Metal Pallet lid at place memory(2)", "Bases at Place Memory" => "Metal Pallet Base at Place", "Clamp Lid" => "Metal Pallet Lid Clamp", "Clamp base" =>, "Move Z" => "Metal Pallet Move Z", "Move X" => "Metal Pallet Move X", Grab => "Metal Pallet Grab", "Pos. raise bases" =>, "Pos. raise lids" => "Metal Pallet pos raise lid", s1 => "Metal  Pallet S1", s2 => "Metal Pallet S2", s3 => "Metal Pallet S3", s4 => "Metal Pallet S4", s5 => "Metal Pallet S5", s6 => "Metal Pallet S6", s7 => "Metal Pallet S7", s8 => "Metal Pallet S8", s9 => "Metal Pallet S9", s10 => "Metal Pallet S10", s11 => "Metal Pallet S11")
   END_RUNG
   // the same network as SCL:
   "Metal Pallet PP"(System := "System",   // "Pick and Place"
                     Start := "Start All Factory",
                     "Lid at place" := "Metal Pallet Lid at Place",
                     "Base at place" := "Metal Pallet Base at Place",
                     "Lid Clamped" := "Metal Pallet Lid Clamped",
                     "Base Clamped" := true,
                     "Item Detected" := "Metal Pallet Item Detected",
                     "Lids Conveyor" => "Metal Pallet Lid Conveyor",
                     "Bases Conveyor" => "Metal Pallet Base Conveyor",
                     "Lids at Place Memory" => "Metal Pallet lid at place memory(2)",
                     "Bases at Place Memory" => "Metal Pallet Base at Place",
                     "Clamp Lid" => "Metal Pallet Lid Clamp",
                     "Move Z" => "Metal Pallet Move Z",
                     "Move X" => "Metal Pallet Move X",
                     Grab => "Metal Pallet Grab",
                     "Pos. raise lids" => "Metal Pallet pos raise lid",
                     s1 => "Metal  Pallet S1",
                     s2 => "Metal Pallet S2",
                     s3 => "Metal Pallet S3",
                     s4 => "Metal Pallet S4",
                     s5 => "Metal Pallet S5",
                     s6 => "Metal Pallet S6",
                     s7 => "Metal Pallet S7",
                     s8 => "Metal Pallet S8",
                     s9 => "Metal Pallet S9",
                     s10 => "Metal Pallet S10",
                     s11 => "Metal Pallet S11");
END_REGION

REGION Network 20
   RUNG wire#powerrail
      "Blue Elevator"("Call Elevator" := "Call Blue Elevator", System := "System", "Elevator Set Point" => "Blue Elevator Set Point", "Elevator Roller" => "Blue Elevator Roller", "Elevator Completed" => "Blue Elevator Completed", "Elevator S1" => "Blue Elevator S1", "Elevator S2" => "Blue Elevator S2", "Elevator S3" => "Blue Elevator S3")
   END_RUNG
   // the same network as SCL:
   "Blue Elevator"("Call Elevator" := "Call Blue Elevator",   // "Elevator"
                   System := "System",
                   "Elevator Set Point" => "Blue Elevator Set Point",
                   "Elevator Roller" => "Blue Elevator Roller",
                   "Elevator Completed" => "Blue Elevator Completed",
                   "Elevator S1" => "Blue Elevator S1",
                   "Elevator S2" => "Blue Elevator S2",
                   "Elevator S3" => "Blue Elevator S3");
END_REGION

REGION Network 21
   RUNG wire#powerrail
      "Green Elevator"("Call Elevator" := "Call Green Elevator", System := "System", "Elevator Set Point" => "Green Elevator Set Point", "Elevator Roller" => "Green Elevator Roller", "Elevator Completed" => "Green Elevator Completed", "Elevator S1" => "Green Elevator S1", "Elevator S2" => "Green Elevator S2", "Elevator S3" => "Green Elevator S3")
   END_RUNG
   // the same network as SCL:
   "Green Elevator"("Call Elevator" := "Call Green Elevator",   // "Elevator"
                    System := "System",
                    "Elevator Set Point" => "Green Elevator Set Point",
                    "Elevator Roller" => "Green Elevator Roller",
                    "Elevator Completed" => "Green Elevator Completed",
                    "Elevator S1" => "Green Elevator S1",
                    "Elevator S2" => "Green Elevator S2",
                    "Elevator S3" => "Green Elevator S3");
END_REGION

REGION Network 22
   RUNG wire#powerrail
      "Metal Elevator"("Call Elevator" := "Call Metal Elevator", System := "System", "Elevator Set Point" => "Metal Elevator Set Point", "Elevator Roller" => "Metal Elevator Roller", "Elevator Completed" => "Metal Elevator Completed", "Elevator S1" => "Metal Elevator S1", "Elevator S2" => "Metal Elevator S2", "Elevator S3" => "Metal Elevator S3")
   END_RUNG
   // the same network as SCL:
   "Metal Elevator"("Call Elevator" := "Call Metal Elevator",   // "Elevator"
                    System := "System",
                    "Elevator Set Point" => "Metal Elevator Set Point",
                    "Elevator Roller" => "Metal Elevator Roller",
                    "Elevator Completed" => "Metal Elevator Completed",
                    "Elevator S1" => "Metal Elevator S1",
                    "Elevator S2" => "Metal Elevator S2",
                    "Elevator S3" => "Metal Elevator S3");
END_REGION

REGION Network 23
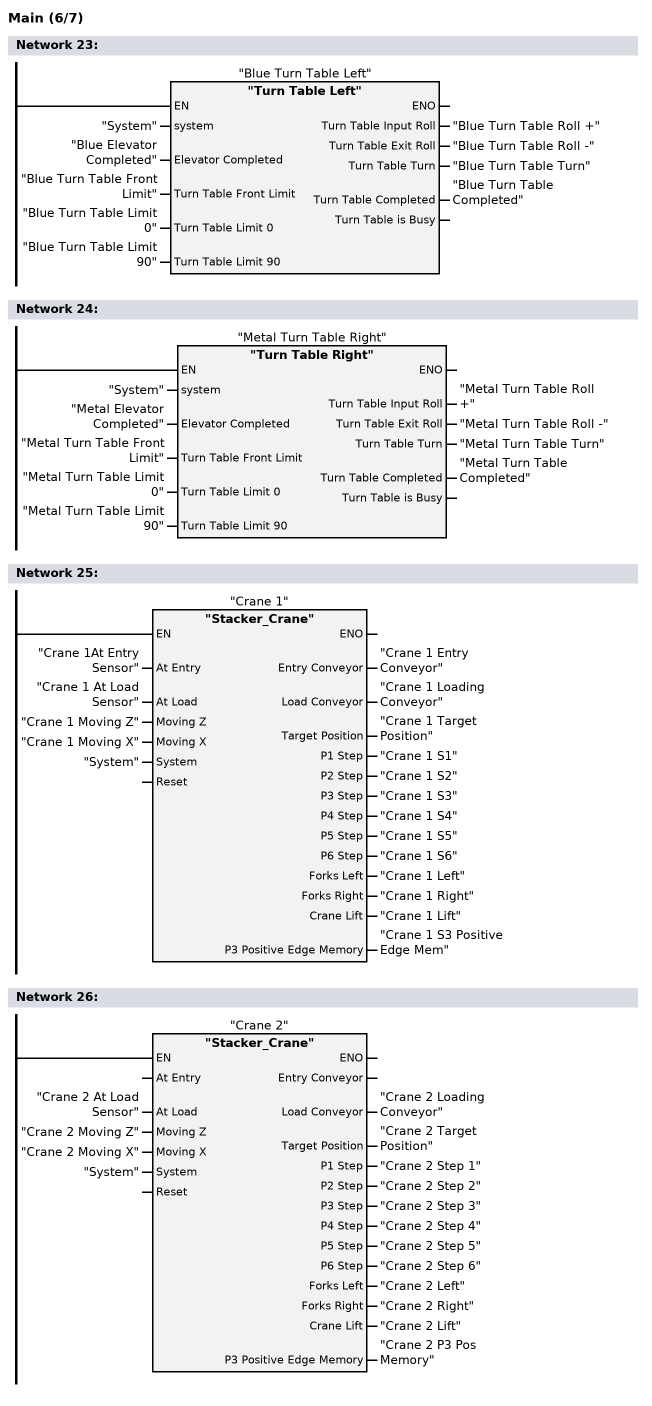
   RUNG wire#powerrail
      "Blue Turn Table Left"(system := "System", "Elevator Completed" := "Blue Elevator Completed", "Turn Table Front Limit" := "Blue Turn Table Front Limit", "Turn Table Limit 0" := "Blue Turn Table Limit 0", "Turn Table Limit 90" := "Blue Turn Table Limit 90", "Turn Table Input Roll" => "Blue Turn Table Roll +", "Turn Table Exit Roll" => "Blue Turn Table Roll -", "Turn Table Turn" => "Blue Turn Table Turn", "Turn Table Completed" => "Blue Turn Table Completed", "Turn Table is Busy" =>)
   END_RUNG
   // the same network as SCL:
   "Blue Turn Table Left"(system := "System",   // "Turn Table Left"
                          "Elevator Completed" := "Blue Elevator Completed",
                          "Turn Table Front Limit" := "Blue Turn Table Front Limit",
                          "Turn Table Limit 0" := "Blue Turn Table Limit 0",
                          "Turn Table Limit 90" := "Blue Turn Table Limit 90",
                          "Turn Table Input Roll" => "Blue Turn Table Roll +",
                          "Turn Table Exit Roll" => "Blue Turn Table Roll -",
                          "Turn Table Turn" => "Blue Turn Table Turn",
                          "Turn Table Completed" => "Blue Turn Table Completed");
END_REGION

REGION Network 24
   RUNG wire#powerrail
      "Metal Turn Table Right"(system := "System", "Elevator Completed" := "Metal Elevator Completed", "Turn Table Front Limit" := "Metal Turn Table Front Limit", "Turn Table Limit 0" := "Metal Turn Table Limit 0", "Turn Table Limit 90" := "Metal Turn Table Limit 90", "Turn Table Input Roll" => "Metal Turn Table Roll +", "Turn Table Exit Roll" => "Metal Turn Table Roll -", "Turn Table Turn" => "Metal Turn Table Turn", "Turn Table Completed" => "Metal Turn Table Completed", "Turn Table is Busy" =>)
   END_RUNG
   // the same network as SCL:
   "Metal Turn Table Right"(system := "System",   // "Turn Table Right"
                           "Elevator Completed" := "Metal Elevator Completed",
                           "Turn Table Front Limit" := "Metal Turn Table Front Limit",
                           "Turn Table Limit 0" := "Metal Turn Table Limit 0",
                           "Turn Table Limit 90" := "Metal Turn Table Limit 90",
                           "Turn Table Input Roll" => "Metal Turn Table Roll +",
                           "Turn Table Exit Roll" => "Metal Turn Table Roll -",
                           "Turn Table Turn" => "Metal Turn Table Turn",
                           "Turn Table Completed" => "Metal Turn Table Completed");
END_REGION

REGION Network 25
   RUNG wire#powerrail
      "Crane 1"("At Entry" := "Crane 1At Entry Sensor", "At Load" := "Crane 1 At Load Sensor", "Moving Z" := "Crane 1 Moving Z", "Moving X" := "Crane 1 Moving X", System := "System", Reset :=, "Entry Conveyor" => "Crane 1 Entry Conveyor", "Load Conveyor" => "Crane 1 Loading Conveyor", "Target Position" => "Crane 1 Target Position", "P1 Step" => "Crane 1 S1", "P2 Step" => "Crane 1 S2", "P3 Step" => "Crane 1 S3", "P4 Step" => "Crane 1 S4", "P5 Step" => "Crane 1 S5", "P6 Step" => "Crane 1 S6", "Forks Left" => "Crane 1 Left", "Forks Right" => "Crane 1 Right", "Crane Lift" => "Crane 1 Lift", "P3 Positive Edge Memory" => "Crane 1 S3 Positive Edge Mem")
   END_RUNG
   // the same network as SCL:
   "Crane 1"("At Entry" := "Crane 1At Entry Sensor",   // "Stacker_Crane"
             "At Load" := "Crane 1 At Load Sensor",
             "Moving Z" := "Crane 1 Moving Z",
             "Moving X" := "Crane 1 Moving X",
             System := "System",
             "Entry Conveyor" => "Crane 1 Entry Conveyor",
             "Load Conveyor" => "Crane 1 Loading Conveyor",
             "Target Position" => "Crane 1 Target Position",
             "P1 Step" => "Crane 1 S1",
             "P2 Step" => "Crane 1 S2",
             "P3 Step" => "Crane 1 S3",
             "P4 Step" => "Crane 1 S4",
             "P5 Step" => "Crane 1 S5",
             "P6 Step" => "Crane 1 S6",
             "Forks Left" => "Crane 1 Left",
             "Forks Right" => "Crane 1 Right",
             "Crane Lift" => "Crane 1 Lift",
             "P3 Positive Edge Memory" => "Crane 1 S3 Positive Edge Mem");
END_REGION

REGION Network 26
   RUNG wire#powerrail
      "Crane 2"("At Entry" :=, "At Load" := "Crane 2 At Load Sensor", "Moving Z" := "Crane 2 Moving Z", "Moving X" := "Crane 2 Moving X", System := "System", Reset :=, "Entry Conveyor" =>, "Load Conveyor" => "Crane 2 Loading Conveyor", "Target Position" => "Crane 2 Target Position", "P1 Step" => "Crane 2 Step 1", "P2 Step" => "Crane 2 Step 2", "P3 Step" => "Crane 2 Step 3", "P4 Step" => "Crane 2 Step 4", "P5 Step" => "Crane 2 Step 5", "P6 Step" => "Crane 2 Step 6", "Forks Left" => "Crane 2 Left", "Forks Right" => "Crane 2 Right", "Crane Lift" => "Crane 2 Lift", "P3 Positive Edge Memory" => "Crane 2 P3 Pos Memory")
   END_RUNG
   // the same network as SCL:
   "Crane 2"("At Load" := "Crane 2 At Load Sensor",   // "Stacker_Crane"
             "Moving Z" := "Crane 2 Moving Z",
             "Moving X" := "Crane 2 Moving X",
             System := "System",
             "Load Conveyor" => "Crane 2 Loading Conveyor",
             "Target Position" => "Crane 2 Target Position",
             "P1 Step" => "Crane 2 Step 1",
             "P2 Step" => "Crane 2 Step 2",
             "P3 Step" => "Crane 2 Step 3",
             "P4 Step" => "Crane 2 Step 4",
             "P5 Step" => "Crane 2 Step 5",
             "P6 Step" => "Crane 2 Step 6",
             "Forks Left" => "Crane 2 Left",
             "Forks Right" => "Crane 2 Right",
             "Crane Lift" => "Crane 2 Lift",
             "P3 Positive Edge Memory" => "Crane 2 P3 Pos Memory");
END_REGION

REGION Network 27
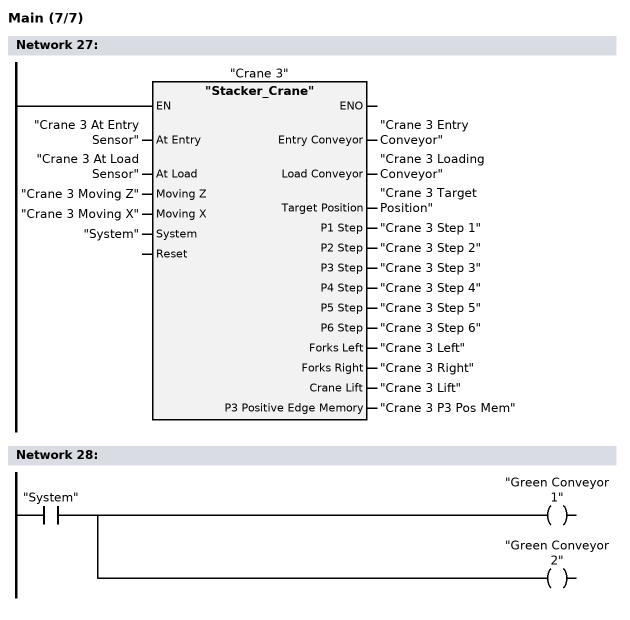
   RUNG wire#powerrail
      "Crane 3"("At Entry" := "Crane 3 At Entry Sensor", "At Load" := "Crane 3 At Load Sensor", "Moving Z" := "Crane 3 Moving Z", "Moving X" := "Crane 3 Moving X", System := "System", Reset :=, "Entry Conveyor" => "Crane 3 Entry Conveyor", "Load Conveyor" => "Crane 3 Loading Conveyor", "Target Position" => "Crane 3 Target Position", "P1 Step" => "Crane 3 Step 1", "P2 Step" => "Crane 3 Step 2", "P3 Step" => "Crane 3 Step 3", "P4 Step" => "Crane 3 Step 4", "P5 Step" => "Crane 3 Step 5", "P6 Step" => "Crane 3 Step 6", "Forks Left" => "Crane 3 Left", "Forks Right" => "Crane 3 Right", "Crane Lift" => "Crane 3 Lift", "P3 Positive Edge Memory" => "Crane 3 P3 Pos Mem")
   END_RUNG
   // the same network as SCL:
   "Crane 3"("At Entry" := "Crane 3 At Entry Sensor",   // "Stacker_Crane"
             "At Load" := "Crane 3 At Load Sensor",
             "Moving Z" := "Crane 3 Moving Z",
             "Moving X" := "Crane 3 Moving X",
             System := "System",
             "Entry Conveyor" => "Crane 3 Entry Conveyor",
             "Load Conveyor" => "Crane 3 Loading Conveyor",
             "Target Position" => "Crane 3 Target Position",
             "P1 Step" => "Crane 3 Step 1",
             "P2 Step" => "Crane 3 Step 2",
             "P3 Step" => "Crane 3 Step 3",
             "P4 Step" => "Crane 3 Step 4",
             "P5 Step" => "Crane 3 Step 5",
             "P6 Step" => "Crane 3 Step 6",
             "Forks Left" => "Crane 3 Left",
             "Forks Right" => "Crane 3 Right",
             "Crane Lift" => "Crane 3 Lift",
             "P3 Positive Edge Memory" => "Crane 3 P3 Pos Mem");
END_REGION

REGION Network 28
   RUNG wire#powerrail
      Contact( "System" )
      wire#w1
      Coil( "Green Conveyor 1" )
   END_RUNG
   RUNG wire#w1
      Coil( "Green Conveyor 2" )
   END_RUNG
   // the same network as SCL:
   "Green Conveyor 1" := "System";
   "Green Conveyor 2" := "System";
END_REGION
END_ORGANIZATION_BLOCK